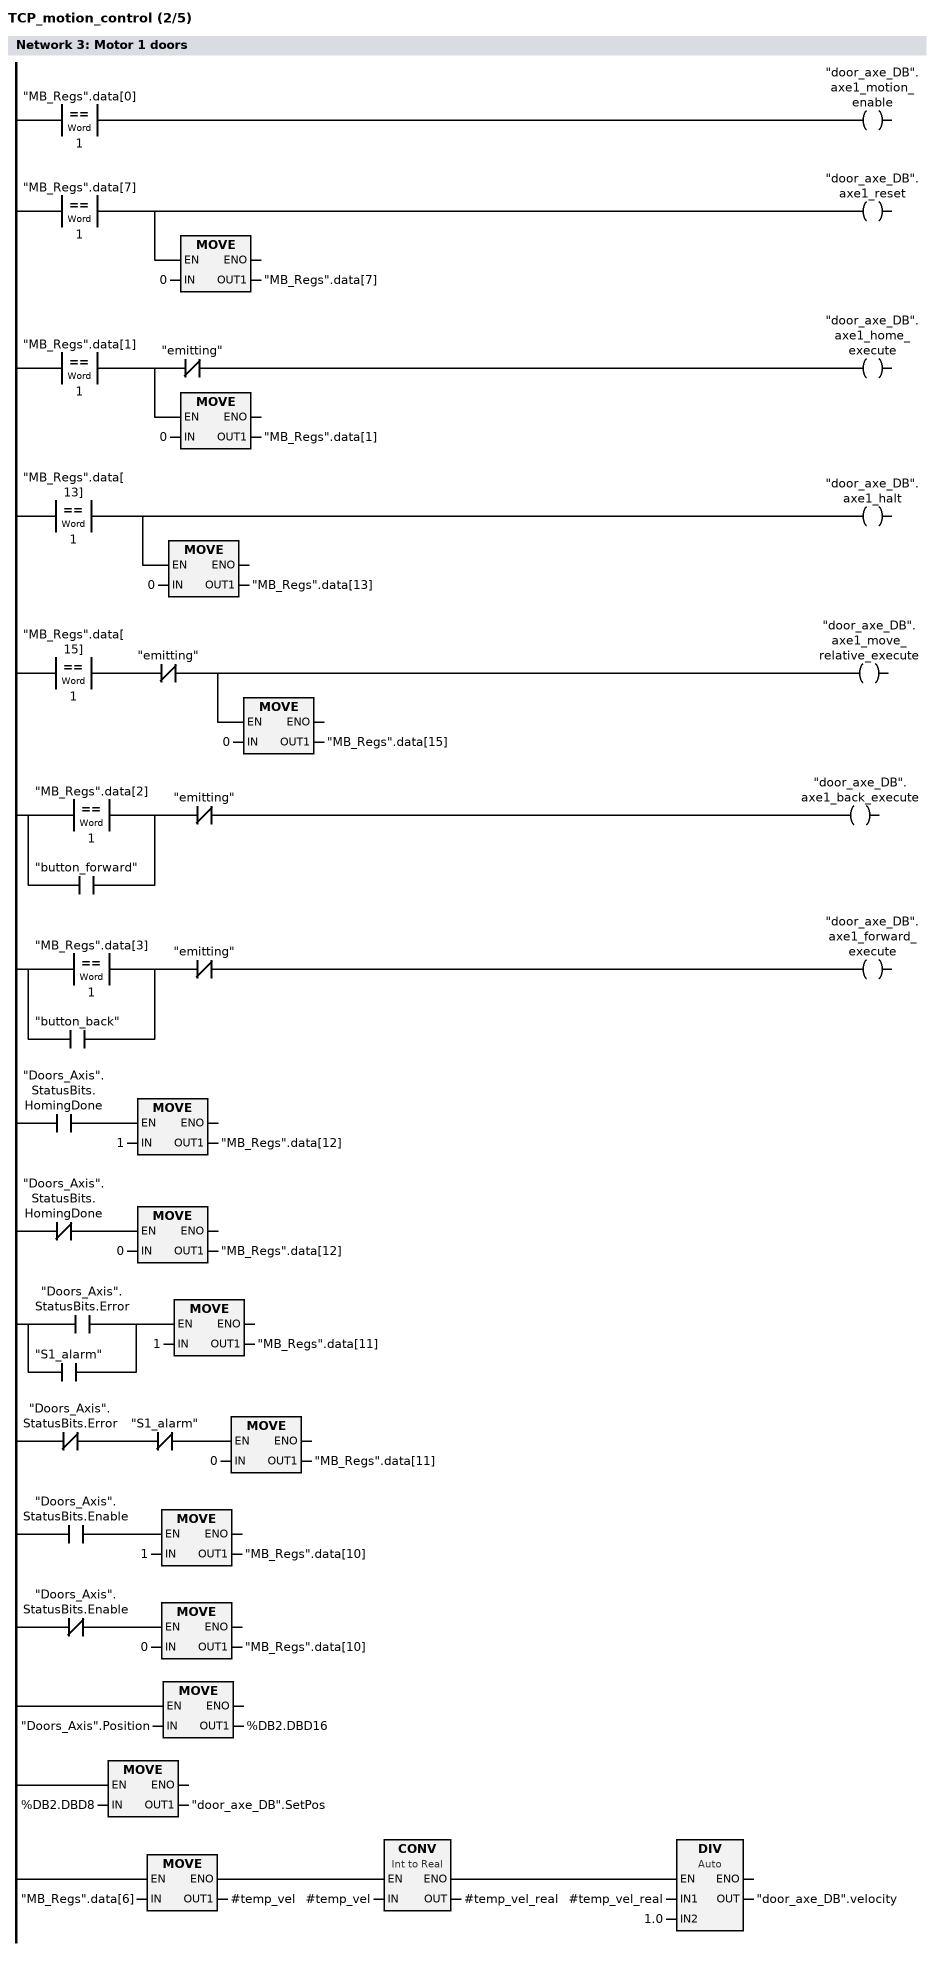
   RUNG wire#powerrail
      { S7_Templates := "SrcType := Word" } EQ_Contact(in1 := "MB_Regs".data[0], in2 := 1)
      Coil( "door_axe_DB".axe1_motion_enable )
   END_RUNG
   RUNG wire#powerrail
      { S7_Templates := "SrcType := Word" } EQ_Contact(in1 := "MB_Regs".data[7], in2 := 1)
      wire#w1
      Coil( "door_axe_DB".axe1_reset )
   END_RUNG
   RUNG wire#w1
      Move(in := 0, out1 => "MB_Regs".data[7])
   END_RUNG
   RUNG wire#powerrail
      { S7_Templates := "SrcType := Word" } EQ_Contact(in1 := "MB_Regs".data[1], in2 := 1)
      wire#w2
      I_Contact( "emitting" )
      Coil( "door_axe_DB".axe1_home_execute )
   END_RUNG
   RUNG wire#w2
      Move(in := 0, out1 => "MB_Regs".data[1])
   END_RUNG
   RUNG wire#powerrail
      { S7_Templates := "SrcType := Word" } EQ_Contact(in1 := "MB_Regs".data[13], in2 := 1)
      wire#w3
      Coil( "door_axe_DB".axe1_halt )
   END_RUNG
   RUNG wire#w3
      Move(in := 0, out1 => "MB_Regs".data[13])
   END_RUNG
   RUNG wire#powerrail
      { S7_Templates := "SrcType := Word" } EQ_Contact(in1 := "MB_Regs".data[15], in2 := 1)
      I_Contact( "emitting" )
      wire#w4
      Coil( "door_axe_DB".axe1_move_relative_execute )
   END_RUNG
   RUNG wire#w4
      Move(in := 0, out1 => "MB_Regs".data[15])
   END_RUNG
   RUNG wire#powerrail
      { S7_Templates := "SrcType := Word" } EQ_Contact(in1 := "MB_Regs".data[2], in2 := 1)
      wire#w5
      I_Contact( "emitting" )
      Coil( "door_axe_DB".axe1_back_execute )
   END_RUNG
   RUNG wire#powerrail
      Contact( "button_forward" )
   END_RUNG wire#w5
   RUNG wire#powerrail
      { S7_Templates := "SrcType := Word" } EQ_Contact(in1 := "MB_Regs".data[3], in2 := 1)
      wire#w6
      I_Contact( "emitting" )
      Coil( "door_axe_DB".axe1_forward_execute )
   END_RUNG
   RUNG wire#powerrail
      Contact( "button_back" )
   END_RUNG wire#w6
   RUNG wire#powerrail
      Contact( "Doors_Axis".StatusBits.HomingDone )
      Move(in := 1, out1 => "MB_Regs".data[12])
   END_RUNG
   RUNG wire#powerrail
      I_Contact( "Doors_Axis".StatusBits.HomingDone )
      Move(in := 0, out1 => "MB_Regs".data[12])
   END_RUNG
   RUNG wire#powerrail
      Contact( "Doors_Axis".StatusBits.Error )
      wire#w7
      Move(in := 1, out1 => "MB_Regs".data[11])
   END_RUNG
   RUNG wire#powerrail
      Contact( "S1_alarm" )
   END_RUNG wire#w7
   RUNG wire#powerrail
      I_Contact( "Doors_Axis".StatusBits.Error )
      I_Contact( "S1_alarm" )
      Move(in := 0, out1 => "MB_Regs".data[11])
   END_RUNG
   RUNG wire#powerrail
      Contact( "Doors_Axis".StatusBits.Enable )
      Move(in := 1, out1 => "MB_Regs".data[10])
   END_RUNG
   RUNG wire#powerrail
      I_Contact( "Doors_Axis".StatusBits.Enable )
      Move(in := 0, out1 => "MB_Regs".data[10])
   END_RUNG
   RUNG wire#powerrail
      Move(in := "Doors_Axis".Position, out1 => %DB2.DBD16)
   END_RUNG
   RUNG wire#powerrail
      Move(in := %DB2.DBD8, out1 => "door_axe_DB".SetPos)
   END_RUNG
   RUNG wire#powerrail
      Move(in := "MB_Regs".data[6], out1 => #temp_vel)
      { S7_Templates := "[SrcType := Int, DestType := Real]" } Convert(in := #temp_vel, out => #temp_vel_real)
      Div(in1 := #temp_vel_real, in2 := 1.0, out => "door_axe_DB".velocity)
   END_RUNG
   // the same network as SCL:
   "door_axe_DB".axe1_motion_enable := "MB_Regs".data[0] = 1;
   "door_axe_DB".axe1_reset := "MB_Regs".data[7] = 1;
   IF "door_axe_DB".axe1_reset THEN "MB_Regs".data[7] := 0; END_IF;
   #_w1 := "MB_Regs".data[1] = 1;
   "door_axe_DB".axe1_home_execute := #_w1 AND NOT "emitting";
   IF #_w1 THEN "MB_Regs".data[1] := 0; END_IF;
   "door_axe_DB".axe1_halt := "MB_Regs".data[13] = 1;
   IF "door_axe_DB".axe1_halt THEN "MB_Regs".data[13] := 0; END_IF;
   "door_axe_DB".axe1_move_relative_execute := ("MB_Regs".data[15] = 1) AND NOT "emitting";
   IF "door_axe_DB".axe1_move_relative_execute THEN "MB_Regs".data[15] := 0; END_IF;
   "door_axe_DB".axe1_back_execute := (("MB_Regs".data[2] = 1) OR "button_forward") AND NOT "emitting";
   "door_axe_DB".axe1_forward_execute := (("MB_Regs".data[3] = 1) OR "button_back") AND NOT "emitting";
   IF "Doors_Axis".StatusBits.HomingDone THEN "MB_Regs".data[12] := 1; END_IF;
   IF NOT "Doors_Axis".StatusBits.HomingDone THEN "MB_Regs".data[12] := 0; END_IF;
   IF "Doors_Axis".StatusBits.Error OR "S1_alarm" THEN "MB_Regs".data[11] := 1; END_IF;
   IF NOT "Doors_Axis".StatusBits.Error AND NOT "S1_alarm" THEN "MB_Regs".data[11] := 0; END_IF;
   IF "Doors_Axis".StatusBits.Enable THEN "MB_Regs".data[10] := 1; END_IF;
   IF NOT "Doors_Axis".StatusBits.Enable THEN "MB_Regs".data[10] := 0; END_IF;
   %DB2.DBD16 := "Doors_Axis".Position;
   "door_axe_DB".SetPos := %DB2.DBD8;
   #temp_vel := "MB_Regs".data[6];
   #temp_vel_real := INT_TO_REAL(#temp_vel);
   "door_axe_DB".velocity := #temp_vel_real / 1.0;
END_REGION

REGION Network 4: Motor 2 rotation
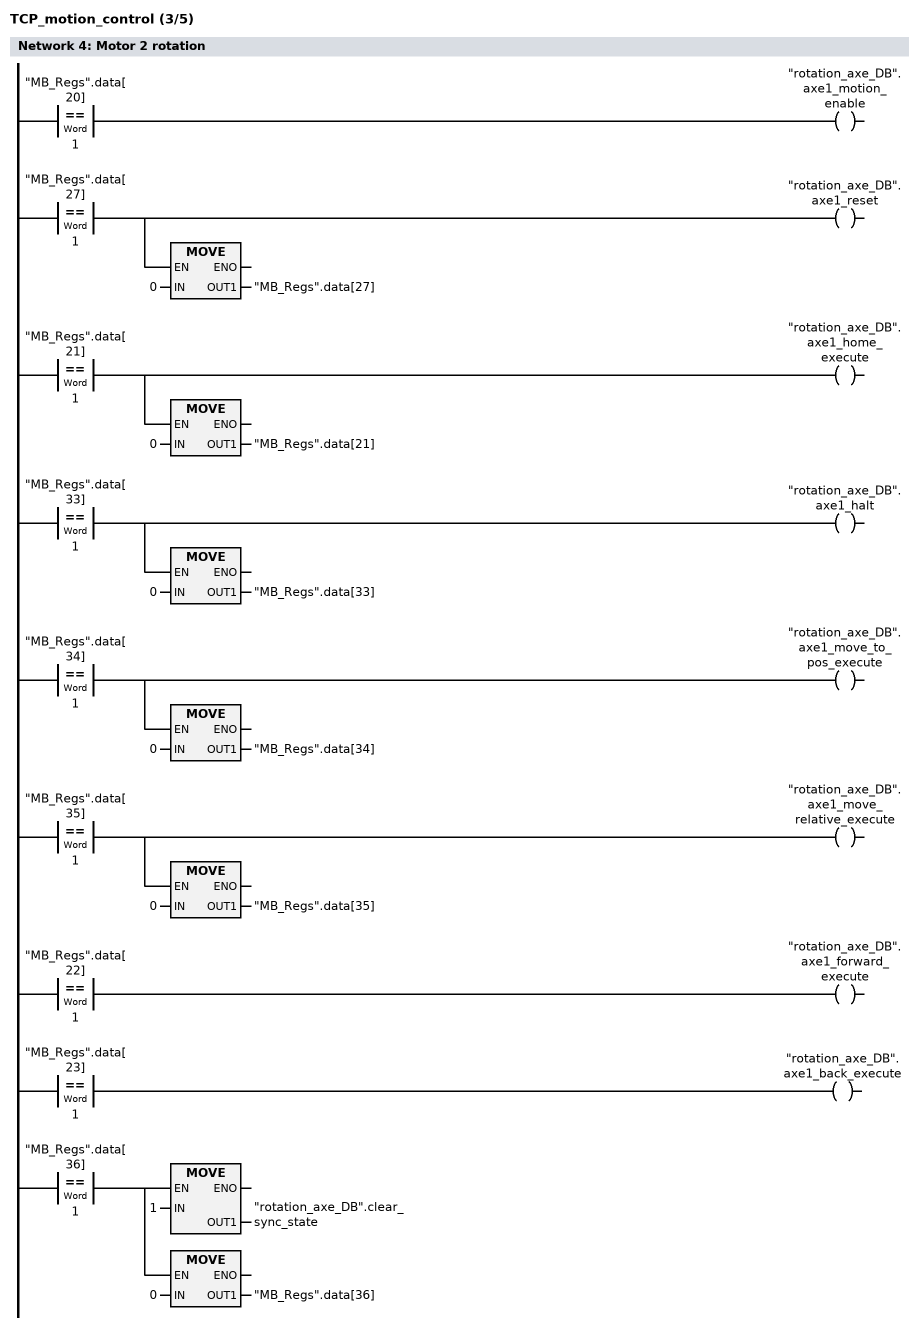
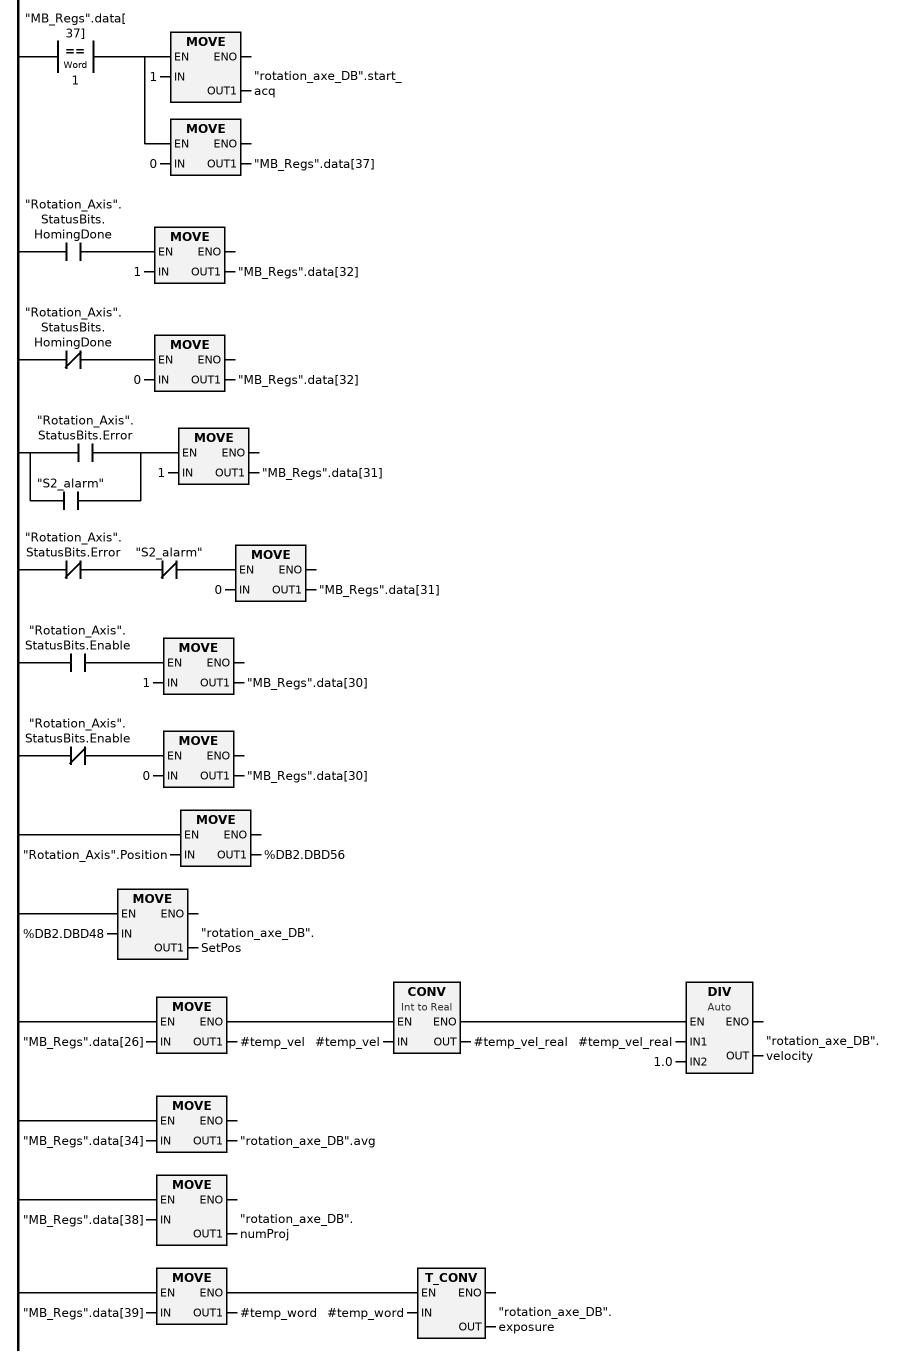
   "rotation_axe_DB".axe1_motion_enable := "MB_Regs".data[20] = 1;
   "rotation_axe_DB".axe1_reset := "MB_Regs".data[27] = 1;
   IF "rotation_axe_DB".axe1_reset THEN "MB_Regs".data[27] := 0; END_IF;
   "rotation_axe_DB".axe1_home_execute := "MB_Regs".data[21] = 1;
   IF "rotation_axe_DB".axe1_home_execute THEN "MB_Regs".data[21] := 0; END_IF;
   "rotation_axe_DB".axe1_halt := "MB_Regs".data[33] = 1;
   IF "rotation_axe_DB".axe1_halt THEN "MB_Regs".data[33] := 0; END_IF;
   "rotation_axe_DB".axe1_move_to_pos_execute := "MB_Regs".data[34] = 1;
   IF "rotation_axe_DB".axe1_move_to_pos_execute THEN "MB_Regs".data[34] := 0; END_IF;
   "rotation_axe_DB".axe1_move_relative_execute := "MB_Regs".data[35] = 1;
   IF "rotation_axe_DB".axe1_move_relative_execute THEN "MB_Regs".data[35] := 0; END_IF;
   "rotation_axe_DB".axe1_forward_execute := "MB_Regs".data[22] = 1;
   "rotation_axe_DB".axe1_back_execute := "MB_Regs".data[23] = 1;
   IF "MB_Regs".data[36] = 1 THEN
       "rotation_axe_DB".clear_sync_state := 1;
       "MB_Regs".data[36] := 0;
   END_IF;
   IF "MB_Regs".data[37] = 1 THEN
       "rotation_axe_DB".start_acq := 1;
       "MB_Regs".data[37] := 0;
   END_IF;
   IF "Rotation_Axis".StatusBits.HomingDone THEN "MB_Regs".data[32] := 1; END_IF;
   IF NOT "Rotation_Axis".StatusBits.HomingDone THEN "MB_Regs".data[32] := 0; END_IF;
   IF "Rotation_Axis".StatusBits.Error OR "S2_alarm" THEN "MB_Regs".data[31] := 1; END_IF;
   IF NOT "Rotation_Axis".StatusBits.Error AND NOT "S2_alarm" THEN "MB_Regs".data[31] := 0; END_IF;
   IF "Rotation_Axis".StatusBits.Enable THEN "MB_Regs".data[30] := 1; END_IF;
   IF NOT "Rotation_Axis".StatusBits.Enable THEN "MB_Regs".data[30] := 0; END_IF;
   %DB2.DBD56 := "Rotation_Axis".Position;
   "rotation_axe_DB".SetPos := %DB2.DBD48;
   #temp_vel := "MB_Regs".data[26];
   #temp_vel_real := INT_TO_REAL(#temp_vel);
   "rotation_axe_DB".velocity := #temp_vel_real / 1.0;
   "rotation_axe_DB".avg := "MB_Regs".data[34];
   "rotation_axe_DB".numProj := "MB_Regs".data[38];
   #temp_word := "MB_Regs".data[39];
   "rotation_axe_DB".exposure := T_CONV(IN := #temp_word);
END_REGION

REGION Network 5: Motor 3 (ISO)
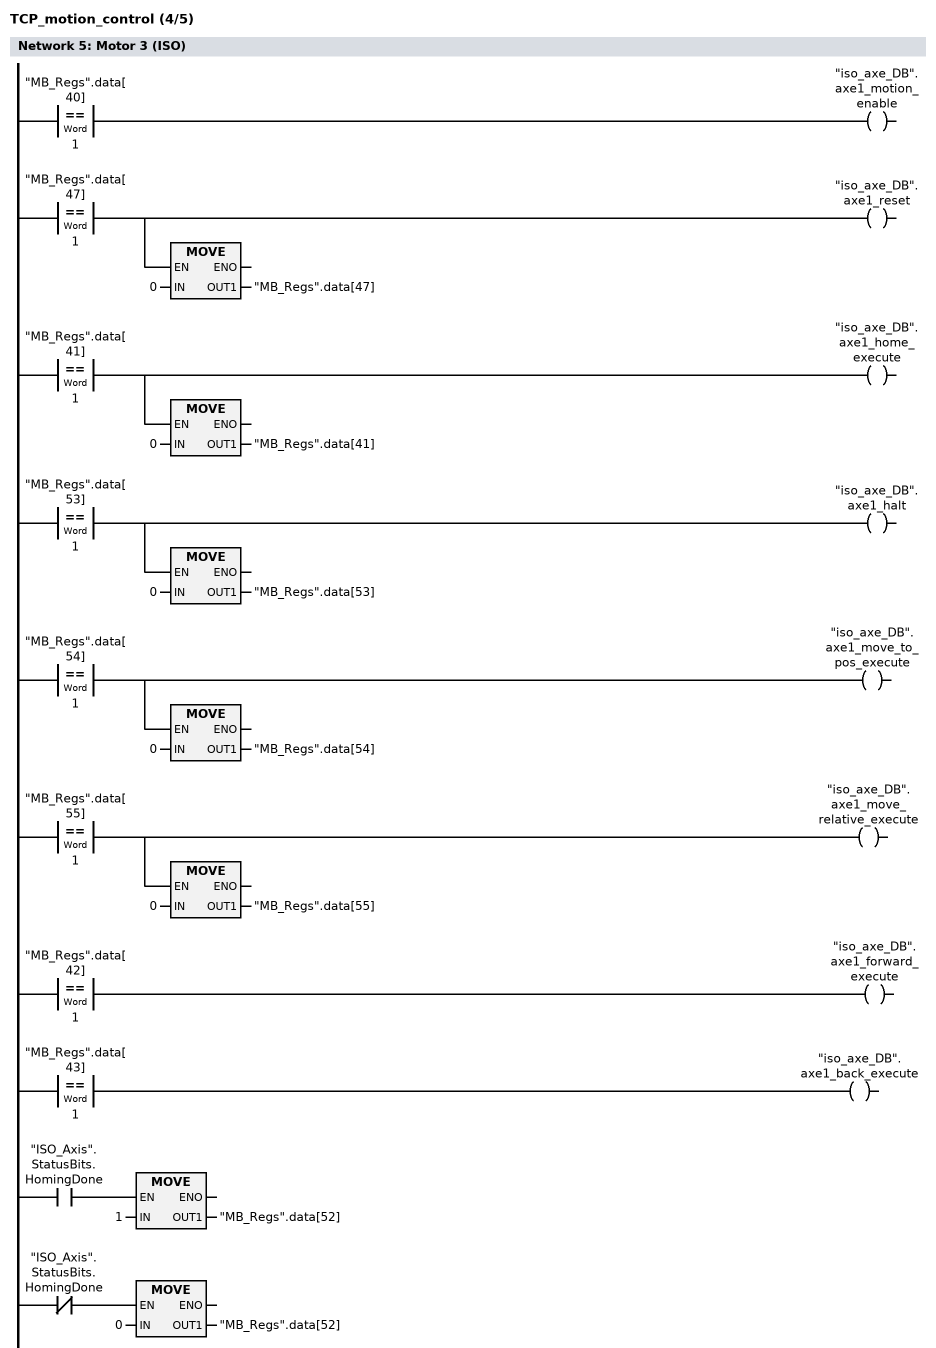
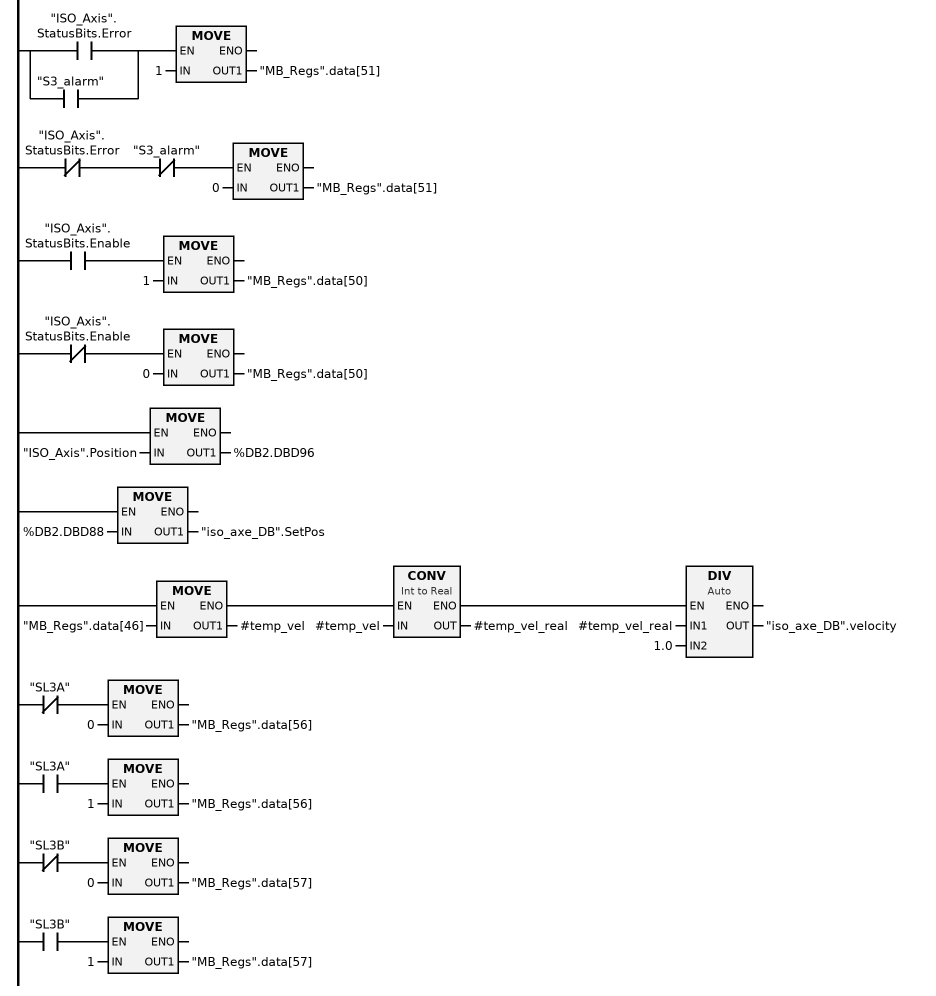
   RUNG wire#powerrail
      { S7_Templates := "SrcType := Word" } EQ_Contact(in1 := "MB_Regs".data[40], in2 := 1)
      Coil( "iso_axe_DB".axe1_motion_enable )
   END_RUNG
   RUNG wire#powerrail
      { S7_Templates := "SrcType := Word" } EQ_Contact(in1 := "MB_Regs".data[47], in2 := 1)
      wire#w1
      Coil( "iso_axe_DB".axe1_reset )
   END_RUNG
   RUNG wire#w1
      Move(in := 0, out1 => "MB_Regs".data[47])
   END_RUNG
   RUNG wire#powerrail
      { S7_Templates := "SrcType := Word" } EQ_Contact(in1 := "MB_Regs".data[41], in2 := 1)
      wire#w2
      Coil( "iso_axe_DB".axe1_home_execute )
   END_RUNG
   RUNG wire#w2
      Move(in := 0, out1 => "MB_Regs".data[41])
   END_RUNG
   RUNG wire#powerrail
      { S7_Templates := "SrcType := Word" } EQ_Contact(in1 := "MB_Regs".data[53], in2 := 1)
      wire#w3
      Coil( "iso_axe_DB".axe1_halt )
   END_RUNG
   RUNG wire#w3
      Move(in := 0, out1 => "MB_Regs".data[53])
   END_RUNG
   RUNG wire#powerrail
      { S7_Templates := "SrcType := Word" } EQ_Contact(in1 := "MB_Regs".data[54], in2 := 1)
      wire#w4
      Coil( "iso_axe_DB".axe1_move_to_pos_execute )
   END_RUNG
   RUNG wire#w4
      Move(in := 0, out1 => "MB_Regs".data[54])
   END_RUNG
   RUNG wire#powerrail
      { S7_Templates := "SrcType := Word" } EQ_Contact(in1 := "MB_Regs".data[55], in2 := 1)
      wire#w5
      Coil( "iso_axe_DB".axe1_move_relative_execute )
   END_RUNG
   RUNG wire#w5
      Move(in := 0, out1 => "MB_Regs".data[55])
   END_RUNG
   RUNG wire#powerrail
      { S7_Templates := "SrcType := Word" } EQ_Contact(in1 := "MB_Regs".data[42], in2 := 1)
      Coil( "iso_axe_DB".axe1_forward_execute )
   END_RUNG
   RUNG wire#powerrail
      { S7_Templates := "SrcType := Word" } EQ_Contact(in1 := "MB_Regs".data[43], in2 := 1)
      Coil( "iso_axe_DB".axe1_back_execute )
   END_RUNG
   RUNG wire#powerrail
      Contact( "ISO_Axis".StatusBits.HomingDone )
      Move(in := 1, out1 => "MB_Regs".data[52])
   END_RUNG
   RUNG wire#powerrail
      I_Contact( "ISO_Axis".StatusBits.HomingDone )
      Move(in := 0, out1 => "MB_Regs".data[52])
   END_RUNG
   RUNG wire#powerrail
      Contact( "ISO_Axis".StatusBits.Error )
      wire#w6
      Move(in := 1, out1 => "MB_Regs".data[51])
   END_RUNG
   RUNG wire#powerrail
      Contact( "S3_alarm" )
   END_RUNG wire#w6
   RUNG wire#powerrail
      I_Contact( "ISO_Axis".StatusBits.Error )
      I_Contact( "S3_alarm" )
      Move(in := 0, out1 => "MB_Regs".data[51])
   END_RUNG
   RUNG wire#powerrail
      Contact( "ISO_Axis".StatusBits.Enable )
      Move(in := 1, out1 => "MB_Regs".data[50])
   END_RUNG
   RUNG wire#powerrail
      I_Contact( "ISO_Axis".StatusBits.Enable )
      Move(in := 0, out1 => "MB_Regs".data[50])
   END_RUNG
   RUNG wire#powerrail
      Move(in := "ISO_Axis".Position, out1 => %DB2.DBD96)
   END_RUNG
   RUNG wire#powerrail
      Move(in := %DB2.DBD88, out1 => "iso_axe_DB".SetPos)
   END_RUNG
   RUNG wire#powerrail
      Move(in := "MB_Regs".data[46], out1 => #temp_vel)
      { S7_Templates := "[SrcType := Int, DestType := Real]" } Convert(in := #temp_vel, out => #temp_vel_real)
      Div(in1 := #temp_vel_real, in2 := 1.0, out => "iso_axe_DB".velocity)
   END_RUNG
   RUNG wire#powerrail
      I_Contact( "SL3A" )
      Move(in := 0, out1 => "MB_Regs".data[56])
   END_RUNG
   RUNG wire#powerrail
      Contact( "SL3A" )
      Move(in := 1, out1 => "MB_Regs".data[56])
   END_RUNG
   RUNG wire#powerrail
      I_Contact( "SL3B" )
      Move(in := 0, out1 => "MB_Regs".data[57])
   END_RUNG
   RUNG wire#powerrail
      Contact( "SL3B" )
      Move(in := 1, out1 => "MB_Regs".data[57])
   END_RUNG
   // the same network as SCL:
   "iso_axe_DB".axe1_motion_enable := "MB_Regs".data[40] = 1;
   "iso_axe_DB".axe1_reset := "MB_Regs".data[47] = 1;
   IF "iso_axe_DB".axe1_reset THEN "MB_Regs".data[47] := 0; END_IF;
   "iso_axe_DB".axe1_home_execute := "MB_Regs".data[41] = 1;
   IF "iso_axe_DB".axe1_home_execute THEN "MB_Regs".data[41] := 0; END_IF;
   "iso_axe_DB".axe1_halt := "MB_Regs".data[53] = 1;
   IF "iso_axe_DB".axe1_halt THEN "MB_Regs".data[53] := 0; END_IF;
   "iso_axe_DB".axe1_move_to_pos_execute := "MB_Regs".data[54] = 1;
   IF "iso_axe_DB".axe1_move_to_pos_execute THEN "MB_Regs".data[54] := 0; END_IF;
   "iso_axe_DB".axe1_move_relative_execute := "MB_Regs".data[55] = 1;
   IF "iso_axe_DB".axe1_move_relative_execute THEN "MB_Regs".data[55] := 0; END_IF;
   "iso_axe_DB".axe1_forward_execute := "MB_Regs".data[42] = 1;
   "iso_axe_DB".axe1_back_execute := "MB_Regs".data[43] = 1;
   IF "ISO_Axis".StatusBits.HomingDone THEN "MB_Regs".data[52] := 1; END_IF;
   IF NOT "ISO_Axis".StatusBits.HomingDone THEN "MB_Regs".data[52] := 0; END_IF;
   IF "ISO_Axis".StatusBits.Error OR "S3_alarm" THEN "MB_Regs".data[51] := 1; END_IF;
   IF NOT "ISO_Axis".StatusBits.Error AND NOT "S3_alarm" THEN "MB_Regs".data[51] := 0; END_IF;
   IF "ISO_Axis".StatusBits.Enable THEN "MB_Regs".data[50] := 1; END_IF;
   IF NOT "ISO_Axis".StatusBits.Enable THEN "MB_Regs".data[50] := 0; END_IF;
   %DB2.DBD96 := "ISO_Axis".Position;
   "iso_axe_DB".SetPos := %DB2.DBD88;
   #temp_vel := "MB_Regs".data[46];
   #temp_vel_real := INT_TO_REAL(#temp_vel);
   "iso_axe_DB".velocity := #temp_vel_real / 1.0;
   IF NOT "SL3A" THEN "MB_Regs".data[56] := 0; END_IF;
   IF "SL3A" THEN "MB_Regs".data[56] := 1; END_IF;
   IF NOT "SL3B" THEN "MB_Regs".data[57] := 0; END_IF;
   IF "SL3B" THEN "MB_Regs".data[57] := 1; END_IF;
END_REGION

REGION Network 6: Motor 4 (Detector)
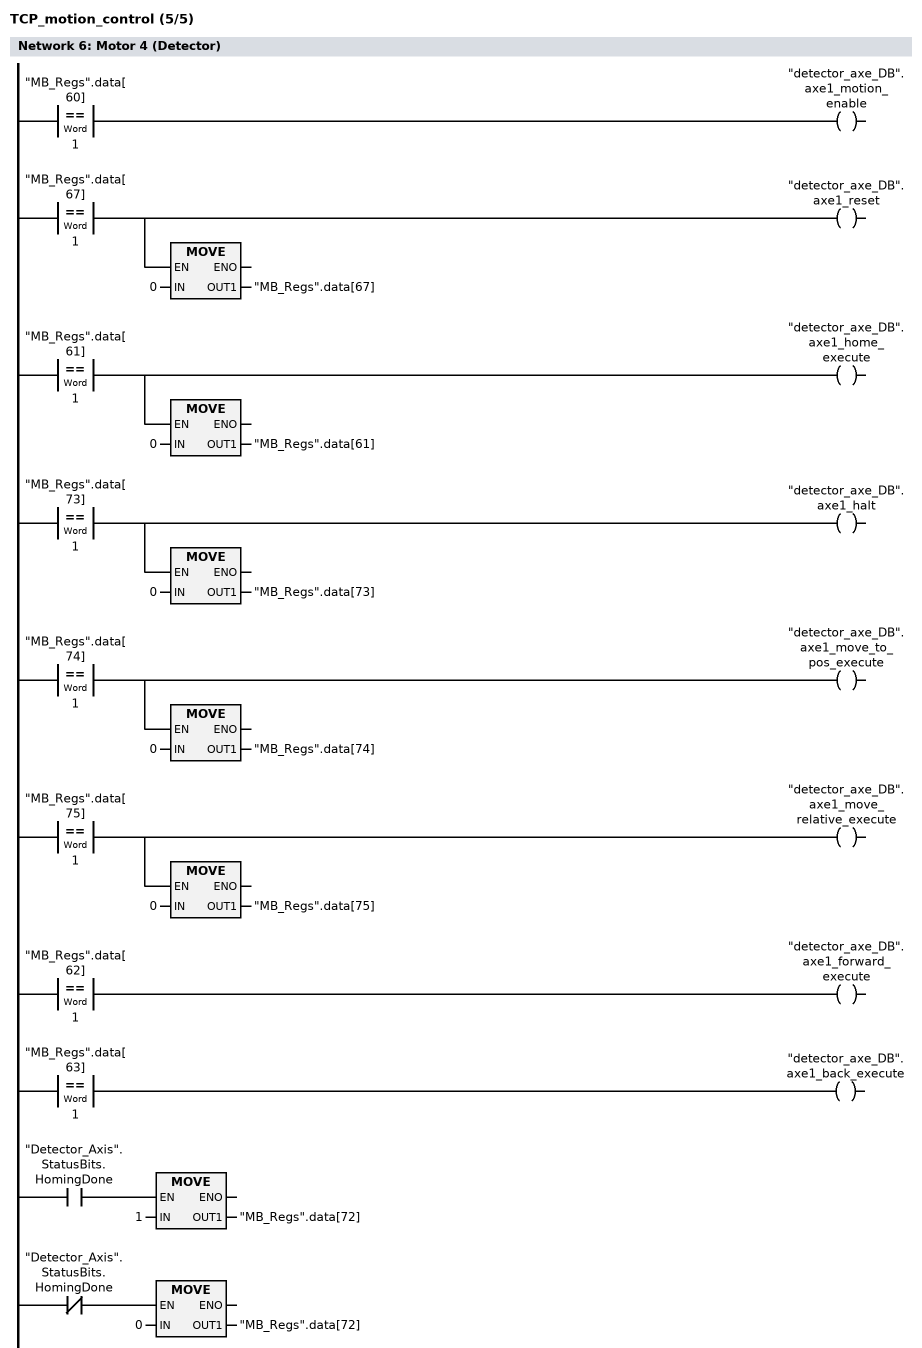
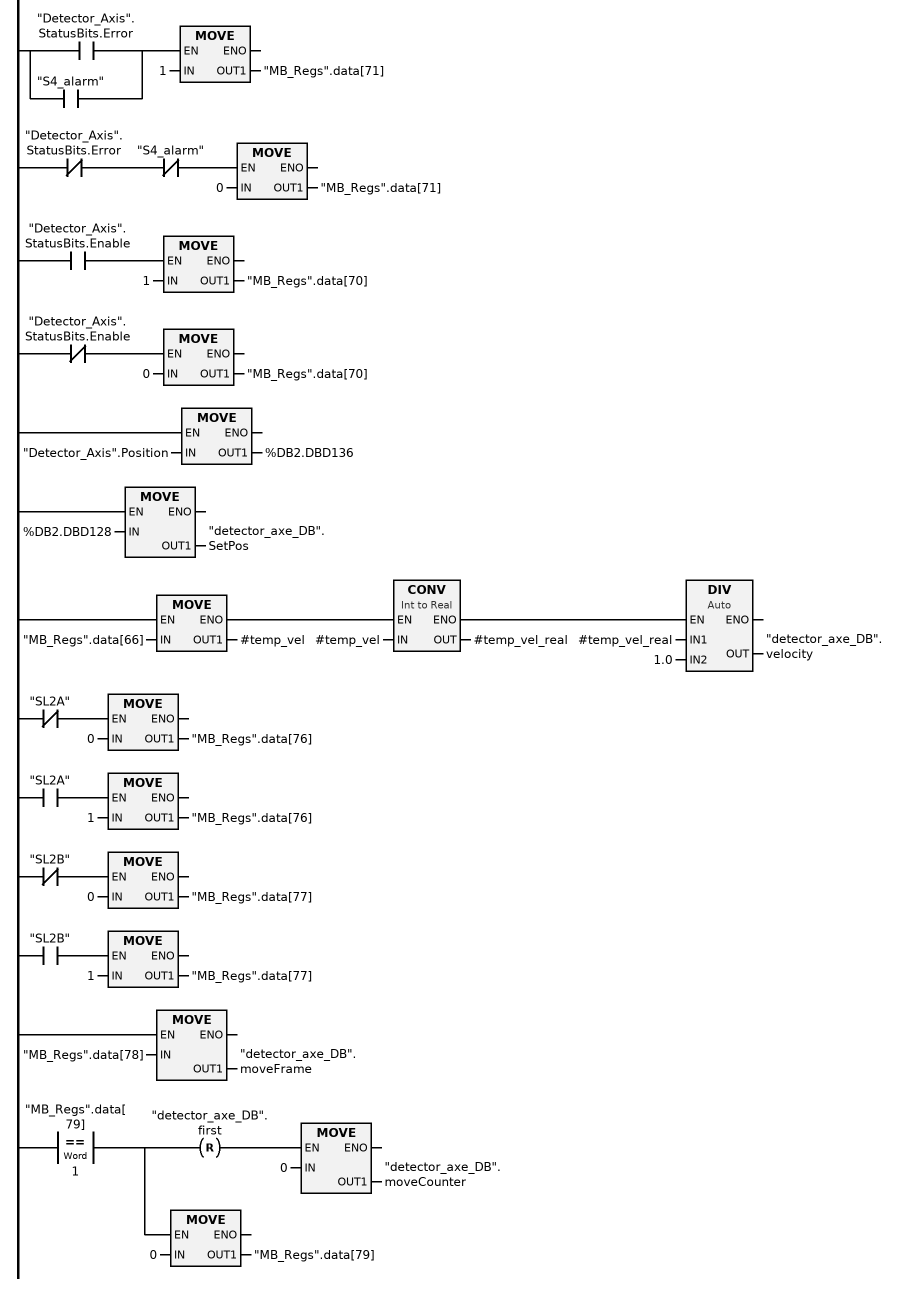
   RUNG wire#powerrail
      { S7_Templates := "SrcType := Word" } EQ_Contact(in1 := "MB_Regs".data[60], in2 := 1)
      Coil( "detector_axe_DB".axe1_motion_enable )
   END_RUNG
   RUNG wire#powerrail
      { S7_Templates := "SrcType := Word" } EQ_Contact(in1 := "MB_Regs".data[67], in2 := 1)
      wire#w1
      Coil( "detector_axe_DB".axe1_reset )
   END_RUNG
   RUNG wire#w1
      Move(in := 0, out1 => "MB_Regs".data[67])
   END_RUNG
   RUNG wire#powerrail
      { S7_Templates := "SrcType := Word" } EQ_Contact(in1 := "MB_Regs".data[61], in2 := 1)
      wire#w2
      Coil( "detector_axe_DB".axe1_home_execute )
   END_RUNG
   RUNG wire#w2
      Move(in := 0, out1 => "MB_Regs".data[61])
   END_RUNG
   RUNG wire#powerrail
      { S7_Templates := "SrcType := Word" } EQ_Contact(in1 := "MB_Regs".data[73], in2 := 1)
      wire#w3
      Coil( "detector_axe_DB".axe1_halt )
   END_RUNG
   RUNG wire#w3
      Move(in := 0, out1 => "MB_Regs".data[73])
   END_RUNG
   RUNG wire#powerrail
      { S7_Templates := "SrcType := Word" } EQ_Contact(in1 := "MB_Regs".data[74], in2 := 1)
      wire#w4
      Coil( "detector_axe_DB".axe1_move_to_pos_execute )
   END_RUNG
   RUNG wire#w4
      Move(in := 0, out1 => "MB_Regs".data[74])
   END_RUNG
   RUNG wire#powerrail
      { S7_Templates := "SrcType := Word" } EQ_Contact(in1 := "MB_Regs".data[75], in2 := 1)
      wire#w5
      Coil( "detector_axe_DB".axe1_move_relative_execute )
   END_RUNG
   RUNG wire#w5
      Move(in := 0, out1 => "MB_Regs".data[75])
   END_RUNG
   RUNG wire#powerrail
      { S7_Templates := "SrcType := Word" } EQ_Contact(in1 := "MB_Regs".data[62], in2 := 1)
      Coil( "detector_axe_DB".axe1_forward_execute )
   END_RUNG
   RUNG wire#powerrail
      { S7_Templates := "SrcType := Word" } EQ_Contact(in1 := "MB_Regs".data[63], in2 := 1)
      Coil( "detector_axe_DB".axe1_back_execute )
   END_RUNG
   RUNG wire#powerrail
      Contact( "Detector_Axis".StatusBits.HomingDone )
      Move(in := 1, out1 => "MB_Regs".data[72])
   END_RUNG
   RUNG wire#powerrail
      I_Contact( "Detector_Axis".StatusBits.HomingDone )
      Move(in := 0, out1 => "MB_Regs".data[72])
   END_RUNG
   RUNG wire#powerrail
      Contact( "Detector_Axis".StatusBits.Error )
      wire#w6
      Move(in := 1, out1 => "MB_Regs".data[71])
   END_RUNG
   RUNG wire#powerrail
      Contact( "S4_alarm" )
   END_RUNG wire#w6
   RUNG wire#powerrail
      I_Contact( "Detector_Axis".StatusBits.Error )
      I_Contact( "S4_alarm" )
      Move(in := 0, out1 => "MB_Regs".data[71])
   END_RUNG
   RUNG wire#powerrail
      Contact( "Detector_Axis".StatusBits.Enable )
      Move(in := 1, out1 => "MB_Regs".data[70])
   END_RUNG
   RUNG wire#powerrail
      I_Contact( "Detector_Axis".StatusBits.Enable )
      Move(in := 0, out1 => "MB_Regs".data[70])
   END_RUNG
   RUNG wire#powerrail
      Move(in := "Detector_Axis".Position, out1 => %DB2.DBD136)
   END_RUNG
   RUNG wire#powerrail
      Move(in := %DB2.DBD128, out1 => "detector_axe_DB".SetPos)
   END_RUNG
   RUNG wire#powerrail
      Move(in := "MB_Regs".data[66], out1 => #temp_vel)
      { S7_Templates := "[SrcType := Int, DestType := Real]" } Convert(in := #temp_vel, out => #temp_vel_real)
      Div(in1 := #temp_vel_real, in2 := 1.0, out => "detector_axe_DB".velocity)
   END_RUNG
   RUNG wire#powerrail
      I_Contact( "SL2A" )
      Move(in := 0, out1 => "MB_Regs".data[76])
   END_RUNG
   RUNG wire#powerrail
      Contact( "SL2A" )
      Move(in := 1, out1 => "MB_Regs".data[76])
   END_RUNG
   RUNG wire#powerrail
      I_Contact( "SL2B" )
      Move(in := 0, out1 => "MB_Regs".data[77])
   END_RUNG
   RUNG wire#powerrail
      Contact( "SL2B" )
      Move(in := 1, out1 => "MB_Regs".data[77])
   END_RUNG
   RUNG wire#powerrail
      Move(in := "MB_Regs".data[78], out1 => "detector_axe_DB".moveFrame)
   END_RUNG
   RUNG wire#powerrail
      { S7_Templates := "SrcType := Word" } EQ_Contact(in1 := "MB_Regs".data[79], in2 := 1)
      wire#w7
      R_Coil( "detector_axe_DB".first )
      Move(in := 0, out1 => "detector_axe_DB".moveCounter)
   END_RUNG
   RUNG wire#w7
      Move(in := 0, out1 => "MB_Regs".data[79])
   END_RUNG
   // the same network as SCL:
   "detector_axe_DB".axe1_motion_enable := "MB_Regs".data[60] = 1;
   "detector_axe_DB".axe1_reset := "MB_Regs".data[67] = 1;
   IF "detector_axe_DB".axe1_reset THEN "MB_Regs".data[67] := 0; END_IF;
   "detector_axe_DB".axe1_home_execute := "MB_Regs".data[61] = 1;
   IF "detector_axe_DB".axe1_home_execute THEN "MB_Regs".data[61] := 0; END_IF;
   "detector_axe_DB".axe1_halt := "MB_Regs".data[73] = 1;
   IF "detector_axe_DB".axe1_halt THEN "MB_Regs".data[73] := 0; END_IF;
   "detector_axe_DB".axe1_move_to_pos_execute := "MB_Regs".data[74] = 1;
   IF "detector_axe_DB".axe1_move_to_pos_execute THEN "MB_Regs".data[74] := 0; END_IF;
   "detector_axe_DB".axe1_move_relative_execute := "MB_Regs".data[75] = 1;
   IF "detector_axe_DB".axe1_move_relative_execute THEN "MB_Regs".data[75] := 0; END_IF;
   "detector_axe_DB".axe1_forward_execute := "MB_Regs".data[62] = 1;
   "detector_axe_DB".axe1_back_execute := "MB_Regs".data[63] = 1;
   IF "Detector_Axis".StatusBits.HomingDone THEN "MB_Regs".data[72] := 1; END_IF;
   IF NOT "Detector_Axis".StatusBits.HomingDone THEN "MB_Regs".data[72] := 0; END_IF;
   IF "Detector_Axis".StatusBits.Error OR "S4_alarm" THEN "MB_Regs".data[71] := 1; END_IF;
   IF NOT "Detector_Axis".StatusBits.Error AND NOT "S4_alarm" THEN "MB_Regs".data[71] := 0; END_IF;
   IF "Detector_Axis".StatusBits.Enable THEN "MB_Regs".data[70] := 1; END_IF;
   IF NOT "Detector_Axis".StatusBits.Enable THEN "MB_Regs".data[70] := 0; END_IF;
   %DB2.DBD136 := "Detector_Axis".Position;
   "detector_axe_DB".SetPos := %DB2.DBD128;
   #temp_vel := "MB_Regs".data[66];
   #temp_vel_real := INT_TO_REAL(#temp_vel);
   "detector_axe_DB".velocity := #temp_vel_real / 1.0;
   IF NOT "SL2A" THEN "MB_Regs".data[76] := 0; END_IF;
   IF "SL2A" THEN "MB_Regs".data[76] := 1; END_IF;
   IF NOT "SL2B" THEN "MB_Regs".data[77] := 0; END_IF;
   IF "SL2B" THEN "MB_Regs".data[77] := 1; END_IF;
   "detector_axe_DB".moveFrame := "MB_Regs".data[78];
   IF "MB_Regs".data[79] = 1 THEN
       "detector_axe_DB".first := FALSE;
       "detector_axe_DB".moveCounter := 0;
       "MB_Regs".data[79] := 0;
   END_IF;
END_REGION
END_FUNCTION_BLOCK

FUNCTION_BLOCK "door_axe"   // FB2, LAD
{ S7_Optimized_Access := 'TRUE' }
VERSION : 0.1
   VAR
      SetPos : Real;
      velocity : Real;
      axe1_motion_enable : Bool;
      axe1_reset : Bool;
      axe1_halt : Bool;
      axe1_forward_execute : Bool;
      axe1_back_execute : Bool;
      axe1_home_execute : Bool;
      axe1_move_to_pos_execute : Bool;
      axe1_move_relative_execute : Bool;
      home_3_busy : Bool;
      home_0_busy : Bool;
      home_3_mode : Bool;
      home_0_mode : Bool;
      axe1_move_done : Bool;
      status : Bool;
   END_VAR
   VAR_TEMP
      temp_val2 : Real;
   END_VAR
   VAR CONSTANT
      vel_const : Real := 2.5;
   END_VAR
   VAR_TEMP   // added for the SCL form of the ladder/FBD networks
      _w1 : Bool;
   END_VAR
BEGIN

REGION Network 1
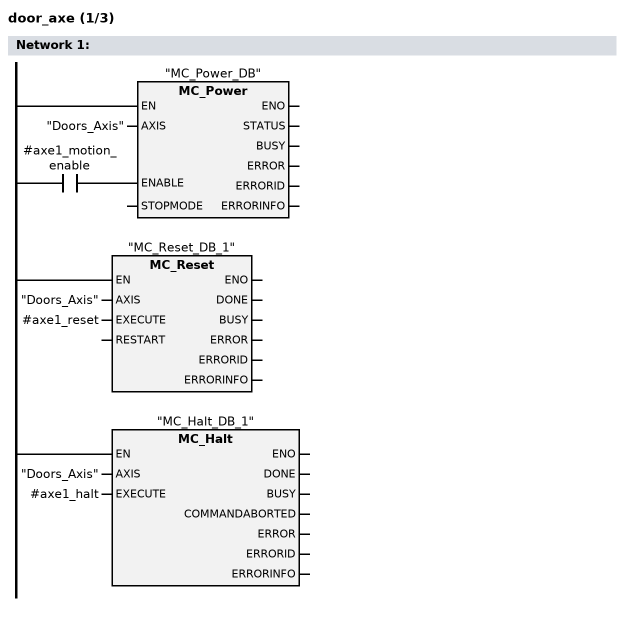
   "MC_Power_DB"(Axis := "Doors_Axis", Enable := #axe1_motion_enable);   // MC_Power
   "MC_Reset_DB_1"(Axis := "Doors_Axis", Execute := #axe1_reset);   // MC_Reset
   "MC_Halt_DB_1"(Axis := "Doors_Axis", Execute := #axe1_halt);   // MC_Halt
END_REGION

REGION Network 2
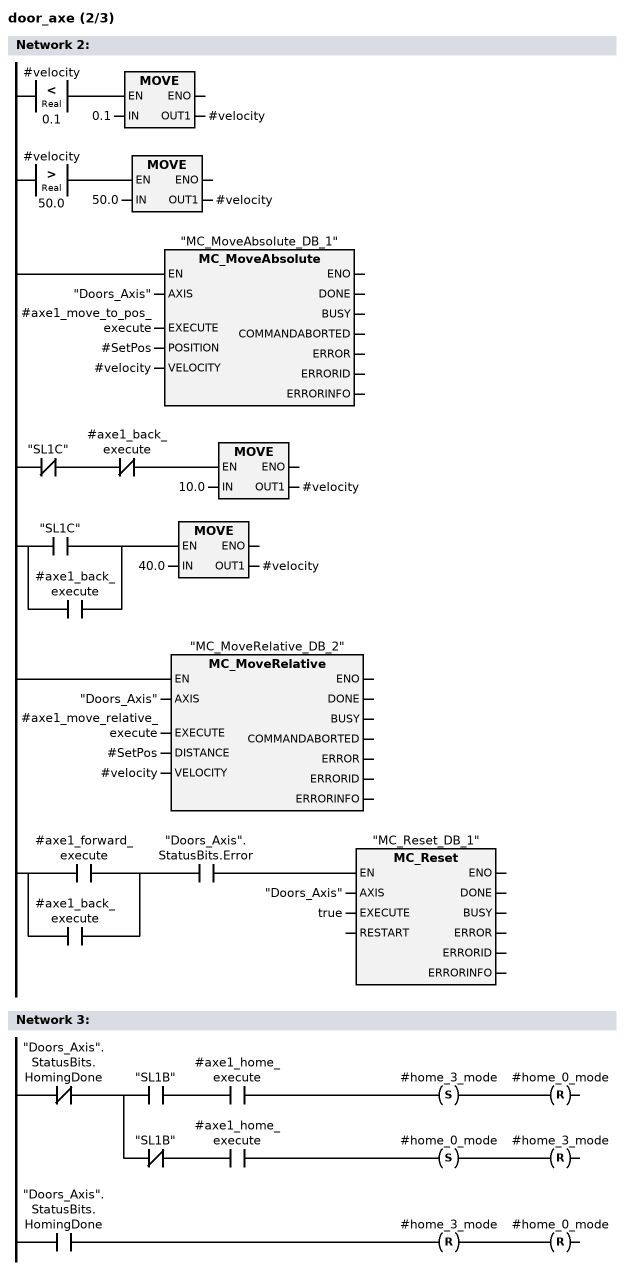
   IF #velocity < 0.1 THEN #velocity := 0.1; END_IF;
   IF #velocity > 50.0 THEN #velocity := 50.0; END_IF;
   "MC_MoveAbsolute_DB_1"(Axis := "Doors_Axis",   // MC_MoveAbsolute
                          Execute := #axe1_move_to_pos_execute,
                          Position := #SetPos,
                          Velocity := #velocity);
   IF NOT "SL1C" AND NOT #axe1_back_execute THEN #velocity := 10.0; END_IF;
   IF "SL1C" OR #axe1_back_execute THEN #velocity := 40.0; END_IF;
   "MC_MoveRelative_DB_2"(Axis := "Doors_Axis",   // MC_MoveRelative
                          Execute := #axe1_move_relative_execute,
                          Distance := #SetPos,
                          Velocity := #velocity);
   IF (#axe1_forward_execute OR #axe1_back_execute) AND "Doors_Axis".StatusBits.Error THEN
       "MC_Reset_DB_1"(Axis := "Doors_Axis", Execute := true);   // MC_Reset
   END_IF;
END_REGION

REGION Network 3
   RUNG wire#powerrail
      I_Contact( "Doors_Axis".StatusBits.HomingDone )
      wire#w1
      Contact( "SL1B" )
      Contact( #axe1_home_execute )
      S_Coil( #home_3_mode )
      R_Coil( #home_0_mode )
   END_RUNG
   RUNG wire#w1
      I_Contact( "SL1B" )
      Contact( #axe1_home_execute )
      S_Coil( #home_0_mode )
      R_Coil( #home_3_mode )
   END_RUNG
   RUNG wire#powerrail
      Contact( "Doors_Axis".StatusBits.HomingDone )
      R_Coil( #home_3_mode )
      R_Coil( #home_0_mode )
   END_RUNG
   // the same network as SCL:
   #_w1 := NOT "Doors_Axis".StatusBits.HomingDone;
   IF #_w1 AND "SL1B" AND #axe1_home_execute THEN
       #home_3_mode := TRUE;
       #home_0_mode := FALSE;
   END_IF;
   IF #_w1 AND NOT "SL1B" AND #axe1_home_execute THEN
       #home_0_mode := TRUE;
       #home_3_mode := FALSE;
   END_IF;
   IF "Doors_Axis".StatusBits.HomingDone THEN
       #home_3_mode := FALSE;
       #home_0_mode := FALSE;
   END_IF;
END_REGION

REGION Network 4: Ручная калибровка
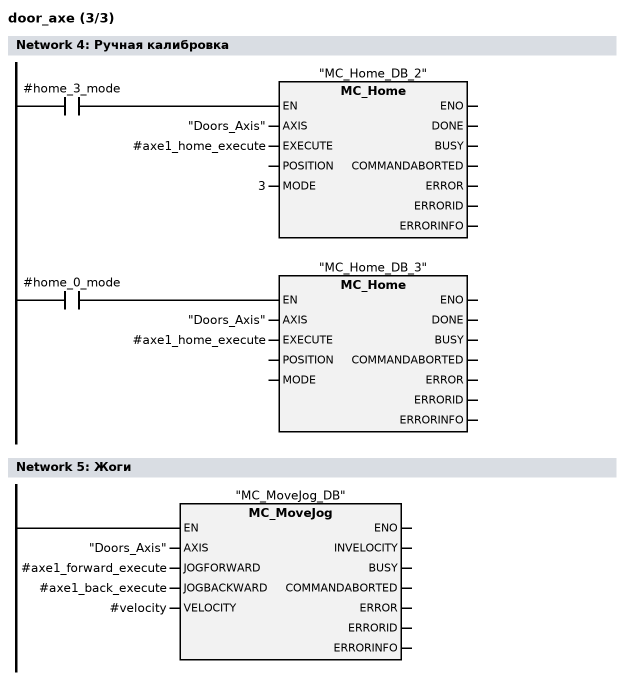
   IF #home_3_mode THEN
       "MC_Home_DB_2"(Axis := "Doors_Axis", Execute := #axe1_home_execute, Mode := 3);   // MC_Home
   END_IF;
   IF #home_0_mode THEN
       "MC_Home_DB_3"(Axis := "Doors_Axis", Execute := #axe1_home_execute);   // MC_Home
   END_IF;
END_REGION

REGION Network 5: Жоги
   "MC_MoveJog_DB"(Axis := "Doors_Axis",   // MC_MoveJog
                   JogForward := #axe1_forward_execute,
                   JogBackward := #axe1_back_execute,
                   Velocity := #velocity);
END_REGION
END_FUNCTION_BLOCK

FUNCTION_BLOCK "rotation_axe"   // FB3, LAD
{ S7_Optimized_Access := 'TRUE' }
VERSION : 0.1
   VAR
      SetPos : Real;
      velocity : Real;
      axe1_motion_enable : Bool;
      axe1_reset : Bool;
      axe1_halt : Bool;
      axe1_forward_execute : Bool;
      axe1_back_execute : Bool;
      axe1_home_execute : Bool;
      axe1_move_to_pos_execute : Bool;
      axe1_move_relative_execute : Bool;
      home_3_busy : Bool;
      home_0_busy : Bool;
      home_3_mode : Bool;
      home_0_mode : Bool;
      axe1_move_done : Bool;
      status : Bool;
      clear_sync_state : Word;
      start_acq : Word;
      projInd : Int;
      numProj : Word;
      exposure : Time;
      avg : Word;
      step1 : Word;
      step2 : Word;
      exposure_phase : Word;
      frd : Word;
      rot : Bool;
      busy : Bool;
      outTime_1 : DTL;
      outTime_12 : DTL;
      retTime_1 : Time;
      outTime_2 : DTL;
      outTime_22 : DTL;
      retTime_2 : Time;
      avgCounter : Word;
      ret : Int;
   END_VAR
   VAR CONSTANT
      vel_const : Real := 2.5;
   END_VAR
   VAR_TEMP   // added for the SCL form of the ladder/FBD networks
      _w1 : Bool;
      _w2 : Bool;
      _w3 : Bool;
      _w4 : Bool;
   END_VAR
BEGIN

REGION Network 1
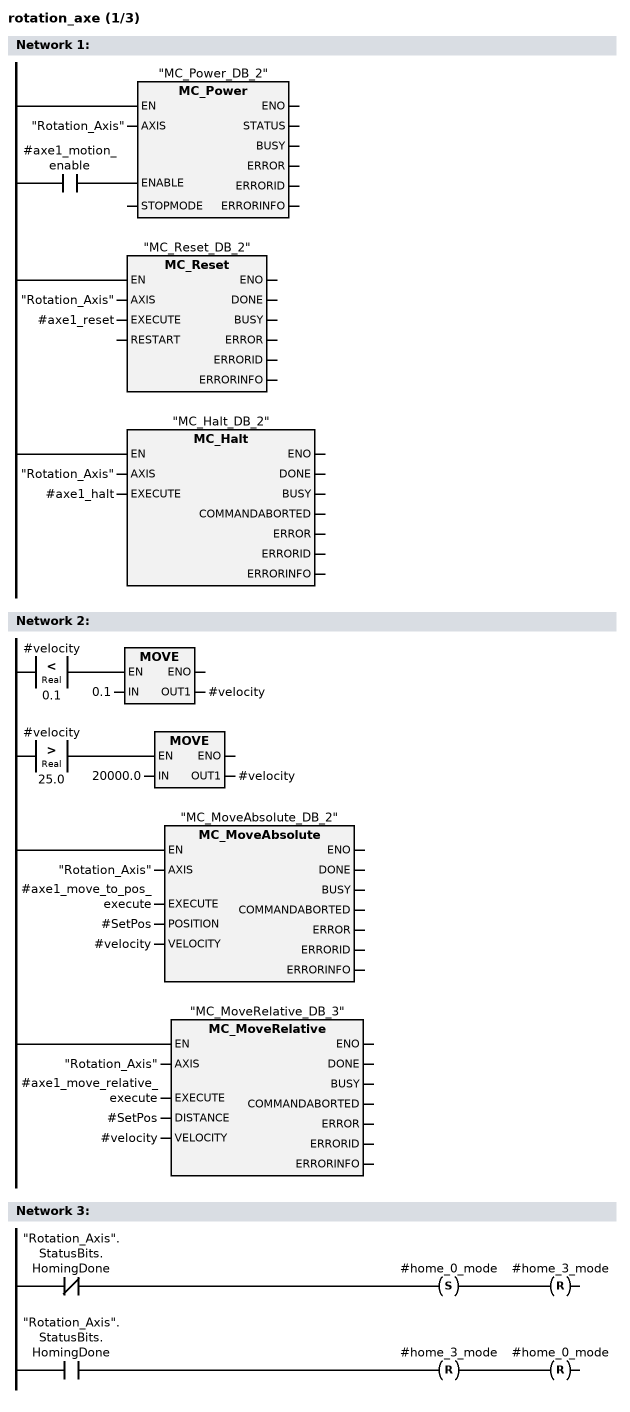
   "MC_Power_DB_2"(Axis := "Rotation_Axis", Enable := #axe1_motion_enable);   // MC_Power
   "MC_Reset_DB_2"(Axis := "Rotation_Axis", Execute := #axe1_reset);   // MC_Reset
   "MC_Halt_DB_2"(Axis := "Rotation_Axis", Execute := #axe1_halt);   // MC_Halt
END_REGION

REGION Network 2
   IF #velocity < 0.1 THEN #velocity := 0.1; END_IF;
   IF #velocity > 25.0 THEN #velocity := 20000.0; END_IF;
   "MC_MoveAbsolute_DB_2"(Axis := "Rotation_Axis",   // MC_MoveAbsolute
                          Execute := #axe1_move_to_pos_execute,
                          Position := #SetPos,
                          Velocity := #velocity);
   "MC_MoveRelative_DB_3"(Axis := "Rotation_Axis",   // MC_MoveRelative
                          Execute := #axe1_move_relative_execute,
                          Distance := #SetPos,
                          Velocity := #velocity);
END_REGION

REGION Network 3
   RUNG wire#powerrail
      I_Contact( "Rotation_Axis".StatusBits.HomingDone )
      S_Coil( #home_0_mode )
      R_Coil( #home_3_mode )
   END_RUNG
   RUNG wire#powerrail
      Contact( "Rotation_Axis".StatusBits.HomingDone )
      R_Coil( #home_3_mode )
      R_Coil( #home_0_mode )
   END_RUNG
   // the same network as SCL:
   IF NOT "Rotation_Axis".StatusBits.HomingDone THEN
       #home_0_mode := TRUE;
       #home_3_mode := FALSE;
   END_IF;
   IF "Rotation_Axis".StatusBits.HomingDone THEN
       #home_3_mode := FALSE;
       #home_0_mode := FALSE;
   END_IF;
END_REGION

REGION Network 4: Ручная калибровка
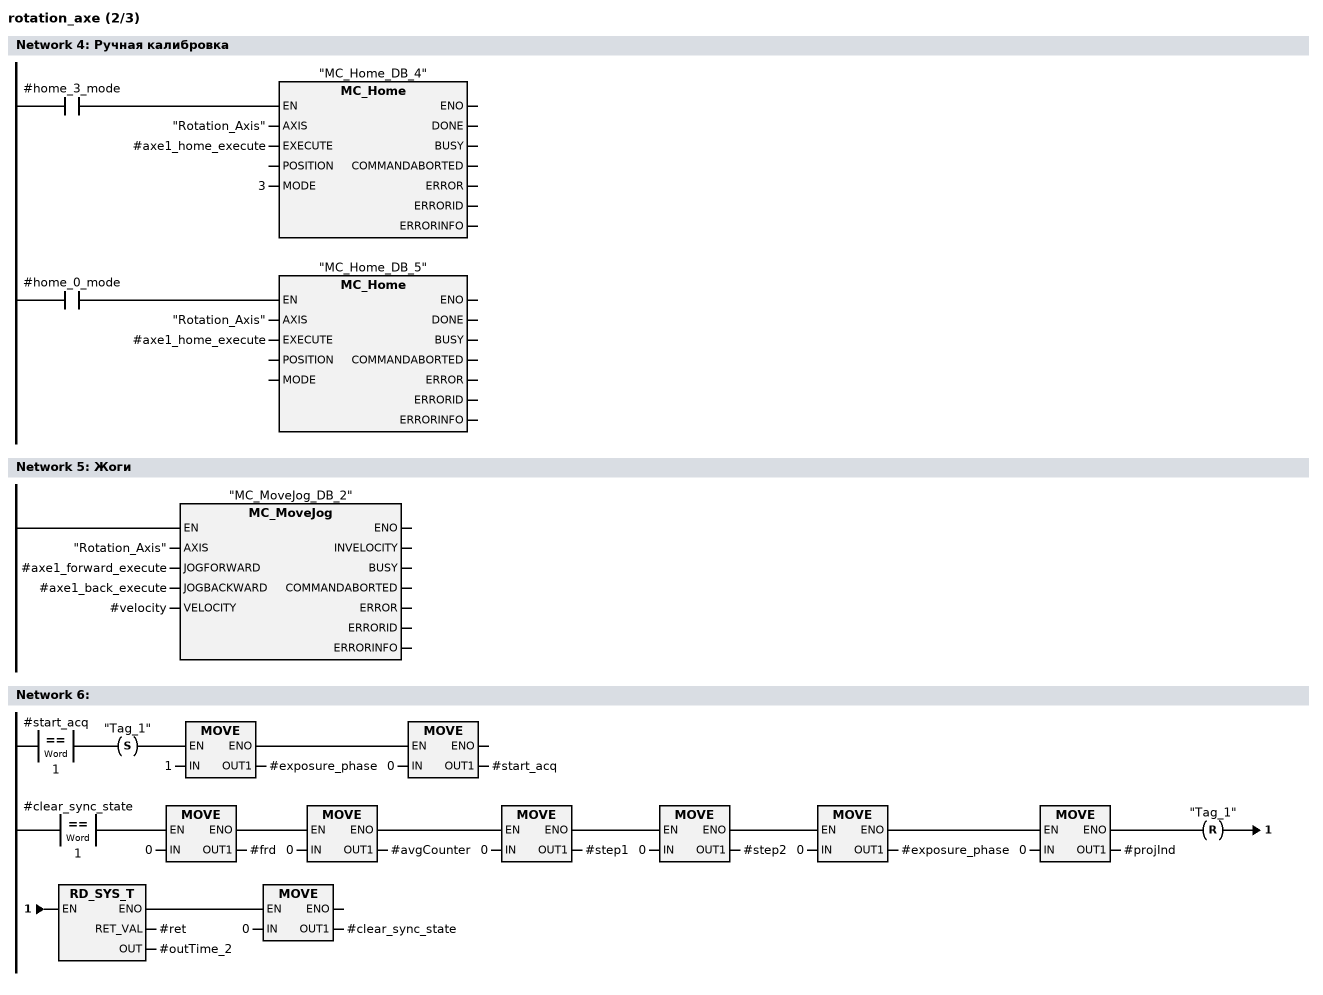
   IF #home_3_mode THEN
       "MC_Home_DB_4"(Axis := "Rotation_Axis", Execute := #axe1_home_execute, Mode := 3);   // MC_Home
   END_IF;
   IF #home_0_mode THEN
       "MC_Home_DB_5"(Axis := "Rotation_Axis", Execute := #axe1_home_execute);   // MC_Home
   END_IF;
END_REGION

REGION Network 5: Жоги
   "MC_MoveJog_DB_2"(Axis := "Rotation_Axis",   // MC_MoveJog
                     JogForward := #axe1_forward_execute,
                     JogBackward := #axe1_back_execute,
                     Velocity := #velocity);
END_REGION

REGION Network 6
   // ENO of a box is taken as its EN; it also drops when the box reports an error
   IF #start_acq = 1 THEN
       "Tag_1" := TRUE;
       #exposure_phase := 1;
       #start_acq := 0;
   END_IF;
   IF #clear_sync_state = 1 THEN
       #frd := 0;
       #avgCounter := 0;
       #step1 := 0;
       #step2 := 0;
       #exposure_phase := 0;
       #projInd := 0;
       "Tag_1" := FALSE;
       #ret := RD_SYS_T(OUT => #outTime_2);
       #clear_sync_state := 0;
   END_IF;
END_REGION

REGION Network 7
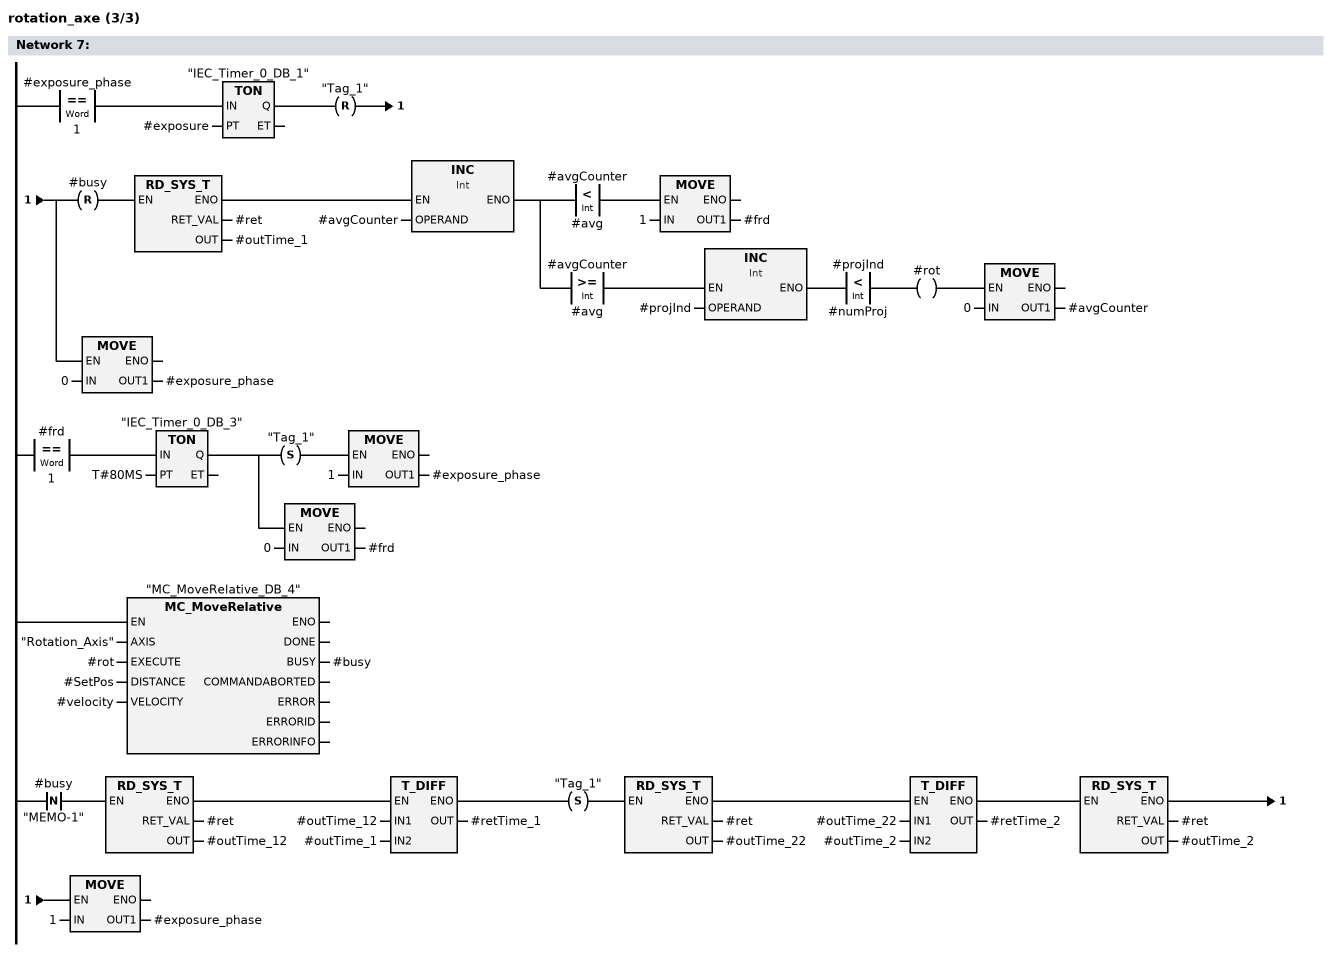
   // ENO of a box is taken as its EN; it also drops when the box reports an error
   "IEC_Timer_0_DB_1".TON(IN := #exposure_phase = 1, PT := #exposure);
   IF "IEC_Timer_0_DB_1".Q THEN
       "Tag_1" := FALSE;
       #busy := FALSE;
   END_IF;
   #_w1 := "IEC_Timer_0_DB_1".Q;
   #_w2 := "IEC_Timer_0_DB_1".Q;
   IF #_w2 THEN
       #ret := RD_SYS_T(OUT => #outTime_1);
       #avgCounter := #avgCounter + 1;
   END_IF;
   IF #_w2 AND (#avgCounter < #avg) THEN #frd := 1; END_IF;
   #_w3 := #_w2 AND (#avgCounter >= #avg);
   IF #_w3 THEN #projInd := #projInd + 1; END_IF;
   #rot := #_w3 AND (#projInd < #numProj);
   IF #rot THEN #avgCounter := 0; END_IF;
   IF #_w1 THEN #exposure_phase := 0; END_IF;
   "IEC_Timer_0_DB_3".TON(IN := #frd = 1, PT := T#80MS);
   IF "IEC_Timer_0_DB_3".Q THEN
       "Tag_1" := TRUE;
       #exposure_phase := 1;
       #frd := 0;
   END_IF;
   "MC_MoveRelative_DB_4"(Axis := "Rotation_Axis",   // MC_MoveRelative
                          Execute := #rot,
                          Distance := #SetPos,
                          Velocity := #velocity,
                          Busy => #busy);
   #_w4 := NOT #busy AND "MEMO-1";   // falling edge of #busy
   "MEMO-1" := #busy;
   IF #_w4 THEN
       #ret := RD_SYS_T(OUT => #outTime_12);
       #retTime_1 := T_DIFF(IN1 := #outTime_12, IN2 := #outTime_1);
       "Tag_1" := TRUE;
       #ret := RD_SYS_T(OUT => #outTime_22);
       #retTime_2 := T_DIFF(IN1 := #outTime_22, IN2 := #outTime_2);
       #ret := RD_SYS_T(OUT => #outTime_2);
       #exposure_phase := 1;
   END_IF;
END_REGION
END_FUNCTION_BLOCK

FUNCTION_BLOCK "detector_axe"   // FB4, LAD
{ S7_Optimized_Access := 'TRUE' }
VERSION : 0.1
   VAR
      SetPos : Real;
      velocity : Real;
      axe1_motion_enable : Bool;
      axe1_reset : Bool;
      axe1_halt : Bool;
      axe1_forward_execute : Bool;
      axe1_back_execute : Bool;
      axe1_home_execute : Bool;
      axe1_move_to_pos_execute : Bool;
      axe1_move_relative_execute : Bool;
      home_3_busy : Bool;
      home_0_busy : Bool;
      home_3_mode : Bool;
      home_0_mode : Bool;
      axe1_move_done : Bool;
      status : Bool;
      moveCounter : Word;
      moveFrame : Word;
      moveCounter2 : Int;
      delayedEx : Bool;
      first : Bool;
   END_VAR
   VAR CONSTANT
      vel_const : Real := 2.5;
   END_VAR
   VAR_TEMP   // added for the SCL form of the ladder/FBD networks
      _w1 : Bool;
      _w2 : Bool;
   END_VAR
BEGIN

REGION Network 1
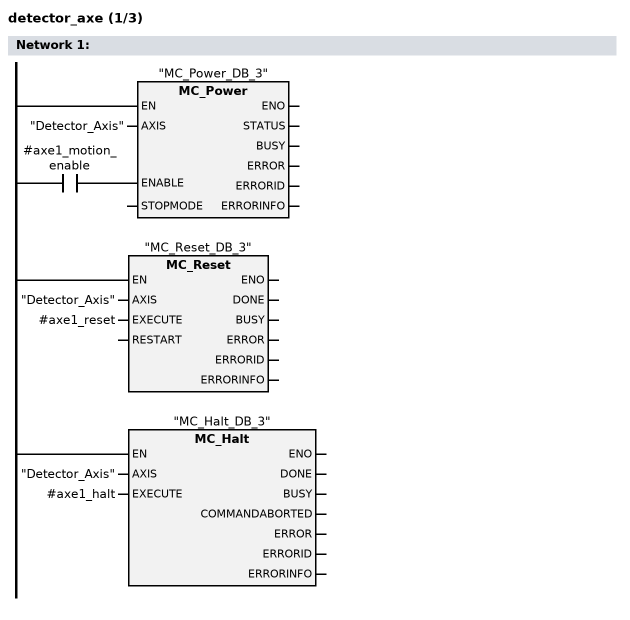
   "MC_Power_DB_3"(Axis := "Detector_Axis", Enable := #axe1_motion_enable);   // MC_Power
   "MC_Reset_DB_3"(Axis := "Detector_Axis", Execute := #axe1_reset);   // MC_Reset
   "MC_Halt_DB_3"(Axis := "Detector_Axis", Execute := #axe1_halt);   // MC_Halt
END_REGION

REGION Network 2
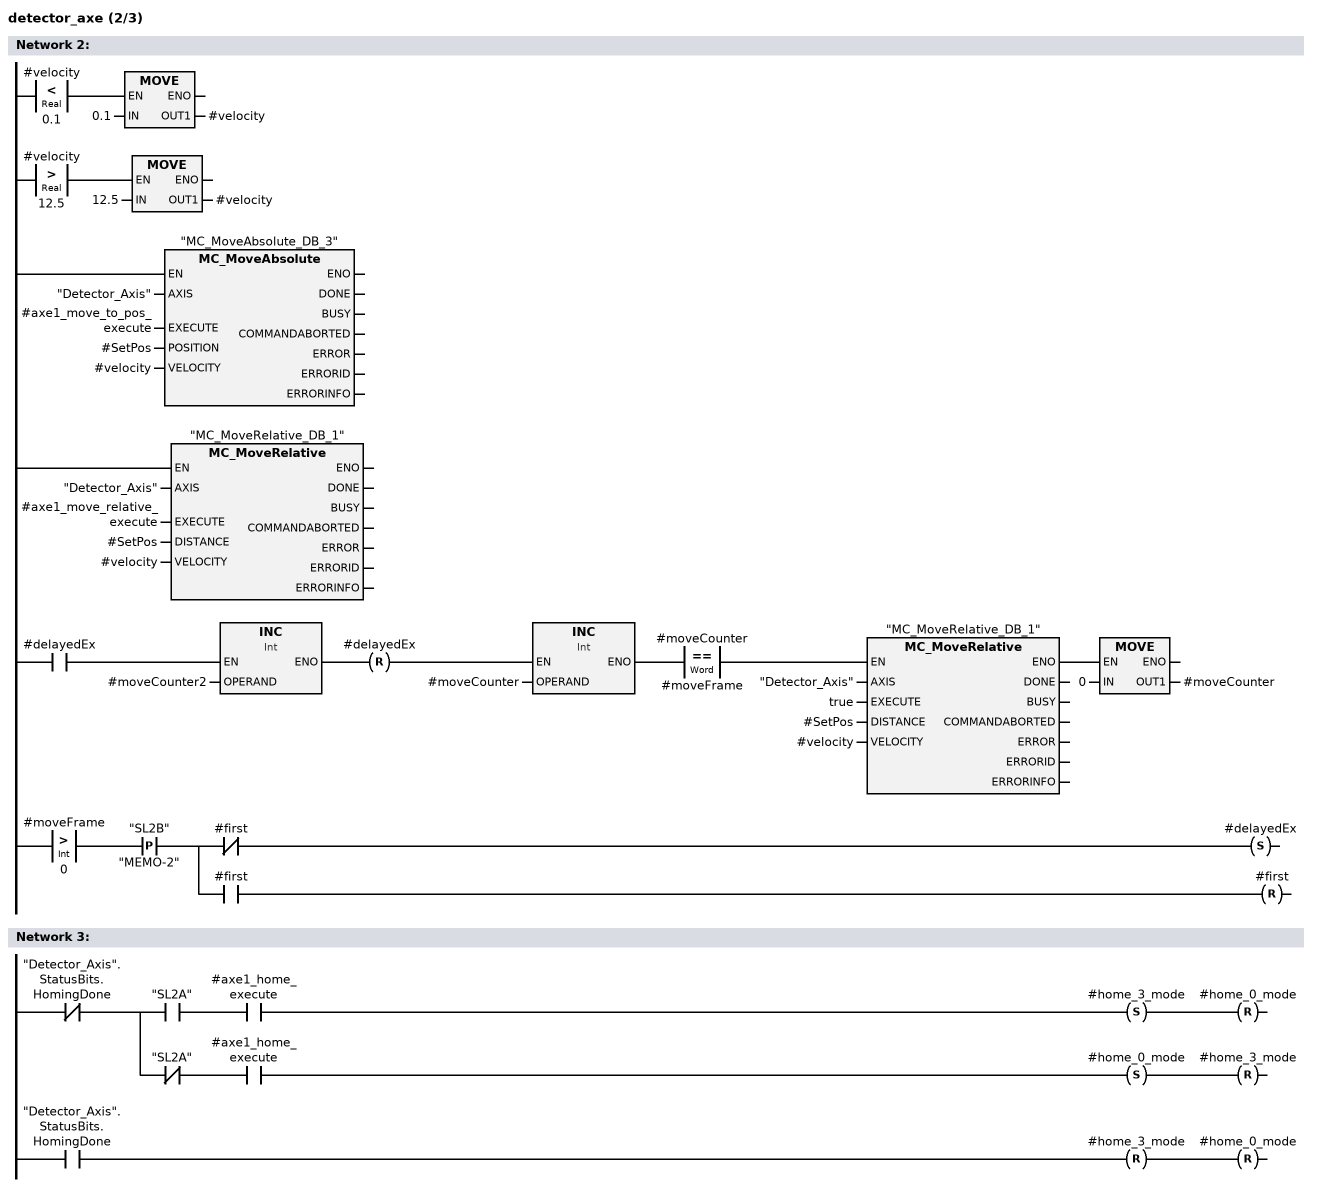
   // ENO of a box is taken as its EN; it also drops when the box reports an error
   IF #velocity < 0.1 THEN #velocity := 0.1; END_IF;
   IF #velocity > 12.5 THEN #velocity := 12.5; END_IF;
   "MC_MoveAbsolute_DB_3"(Axis := "Detector_Axis",   // MC_MoveAbsolute
                          Execute := #axe1_move_to_pos_execute,
                          Position := #SetPos,
                          Velocity := #velocity);
   "MC_MoveRelative_DB_1"(Axis := "Detector_Axis",   // MC_MoveRelative
                          Execute := #axe1_move_relative_execute,
                          Distance := #SetPos,
                          Velocity := #velocity);
   IF #delayedEx THEN #moveCounter2 := #moveCounter2 + 1; END_IF;
   #_w1 := #delayedEx;
   IF #_w1 THEN
       #delayedEx := FALSE;
       #moveCounter := #moveCounter + 1;
   END_IF;
   IF #_w1 AND (#moveCounter = #moveFrame) THEN
       "MC_MoveRelative_DB_1"(Axis := "Detector_Axis", Execute := true, Distance := #SetPos, Velocity := #velocity);   // MC_MoveRelative
       #moveCounter := 0;
   END_IF;
   #_w2 := (#moveFrame > 0) AND "SL2B" AND NOT "MEMO-2";   // rising edge of "SL2B"
   "MEMO-2" := "SL2B";
   IF #_w2 AND NOT #first THEN #delayedEx := TRUE; END_IF;
   IF #_w2 AND #first THEN #first := FALSE; END_IF;
END_REGION

REGION Network 3
   RUNG wire#powerrail
      I_Contact( "Detector_Axis".StatusBits.HomingDone )
      wire#w1
      Contact( "SL2A" )
      Contact( #axe1_home_execute )
      S_Coil( #home_3_mode )
      R_Coil( #home_0_mode )
   END_RUNG
   RUNG wire#w1
      I_Contact( "SL2A" )
      Contact( #axe1_home_execute )
      S_Coil( #home_0_mode )
      R_Coil( #home_3_mode )
   END_RUNG
   RUNG wire#powerrail
      Contact( "Detector_Axis".StatusBits.HomingDone )
      R_Coil( #home_3_mode )
      R_Coil( #home_0_mode )
   END_RUNG
   // the same network as SCL:
   #_w1 := NOT "Detector_Axis".StatusBits.HomingDone;
   IF #_w1 AND "SL2A" AND #axe1_home_execute THEN
       #home_3_mode := TRUE;
       #home_0_mode := FALSE;
   END_IF;
   IF #_w1 AND NOT "SL2A" AND #axe1_home_execute THEN
       #home_0_mode := TRUE;
       #home_3_mode := FALSE;
   END_IF;
   IF "Detector_Axis".StatusBits.HomingDone THEN
       #home_3_mode := FALSE;
       #home_0_mode := FALSE;
   END_IF;
END_REGION

REGION Network 4: Ручная калибровка
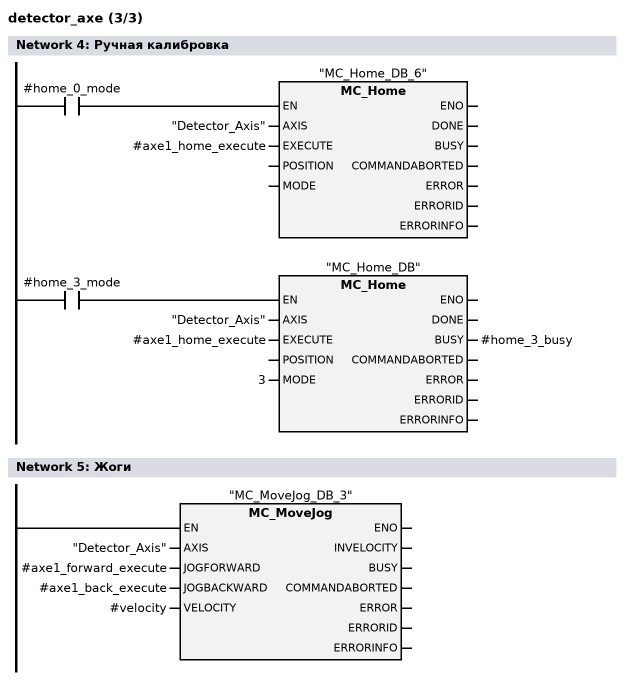
   IF #home_0_mode THEN
       "MC_Home_DB_6"(Axis := "Detector_Axis", Execute := #axe1_home_execute);   // MC_Home
   END_IF;
   IF #home_3_mode THEN
       "MC_Home_DB"(Axis := "Detector_Axis", Execute := #axe1_home_execute, Mode := 3, Busy => #home_3_busy);   // MC_Home
   END_IF;
END_REGION

REGION Network 5: Жоги
   "MC_MoveJog_DB_3"(Axis := "Detector_Axis",   // MC_MoveJog
                     JogForward := #axe1_forward_execute,
                     JogBackward := #axe1_back_execute,
                     Velocity := #velocity);
END_REGION
END_FUNCTION_BLOCK

FUNCTION_BLOCK "safety"   // FB5, LAD
{ S7_Optimized_Access := 'TRUE' }
VERSION : 0.1
BEGIN

REGION Network 1: блокировка излучекеия при открытом периметри
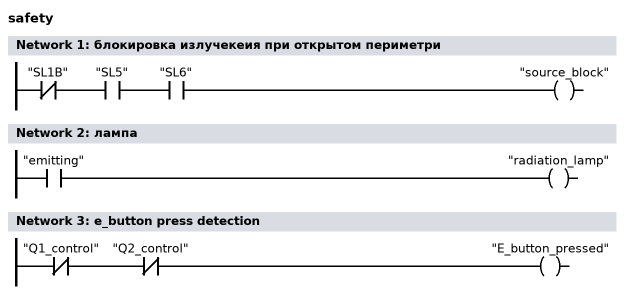
   RUNG wire#powerrail
      I_Contact( "SL1B" )
      Contact( "SL5" )
      Contact( "SL6" )
      Coil( "source_block" )
   END_RUNG
   // the same network as SCL:
   "source_block" := NOT "SL1B" AND "SL5" AND "SL6";
END_REGION

REGION Network 2: лампа
   RUNG wire#powerrail
      Contact( "emitting" )
      Coil( "radiation_lamp" )
   END_RUNG
   // the same network as SCL:
   "radiation_lamp" := "emitting";
END_REGION

REGION Network 3: e_button press detection
   RUNG wire#powerrail
      I_Contact( "Q1_control" )
      I_Contact( "Q2_control" )
      Coil( "E_button_pressed" )
   END_RUNG
   // the same network as SCL:
   "E_button_pressed" := NOT "Q1_control" AND NOT "Q2_control";
END_REGION
END_FUNCTION_BLOCK

FUNCTION_BLOCK "iso_axe"   // FB12, LAD
{ S7_Optimized_Access := 'TRUE' }
VERSION : 0.1
   VAR
      SetPos : Real;
      velocity : Real;
      axe1_motion_enable : Bool;
      axe1_reset : Bool;
      axe1_halt : Bool;
      axe1_forward_execute : Bool;
      axe1_back_execute : Bool;
      axe1_home_execute : Bool;
      axe1_move_to_pos_execute : Bool;
      axe1_move_relative_execute : Bool;
      home_3_busy : Bool;
      home_0_busy : Bool;
      home_3_mode : Bool;
      home_0_mode : Bool;
      axe1_move_done : Bool;
      status : Bool;
   END_VAR
   VAR CONSTANT
      vel_const : Real := 2.5;
   END_VAR
   VAR_TEMP   // added for the SCL form of the ladder/FBD networks
      _w1 : Bool;
   END_VAR
BEGIN

REGION Network 1
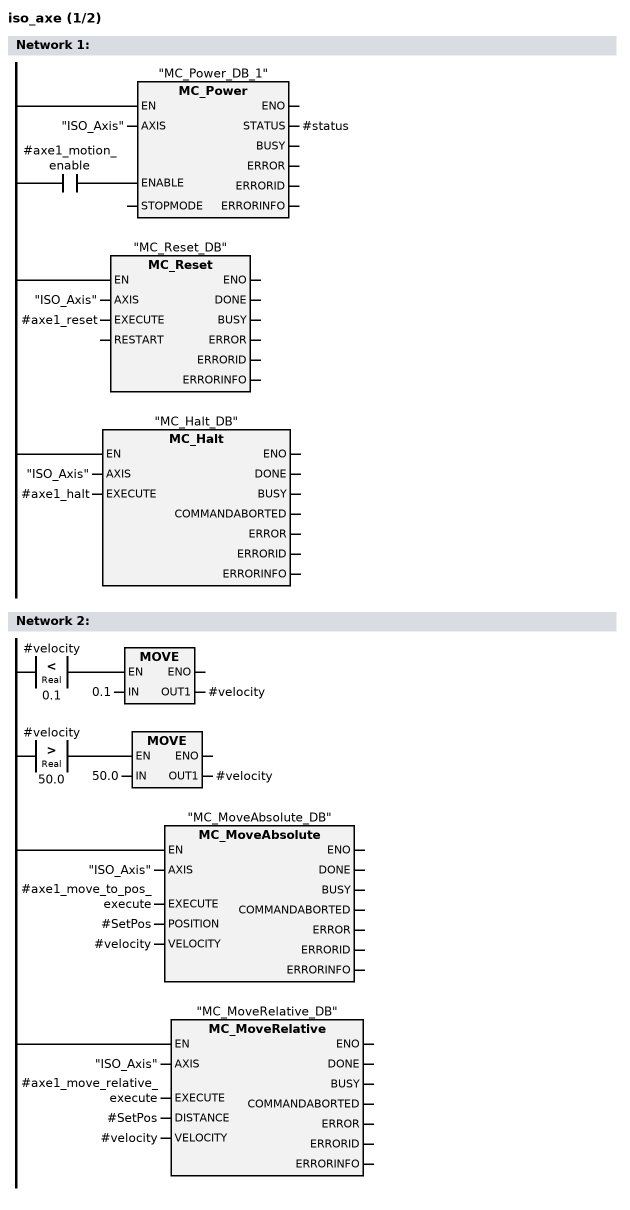
   "MC_Power_DB_1"(Axis := "ISO_Axis", Enable := #axe1_motion_enable, Status => #status);   // MC_Power
   "MC_Reset_DB"(Axis := "ISO_Axis", Execute := #axe1_reset);   // MC_Reset
   "MC_Halt_DB"(Axis := "ISO_Axis", Execute := #axe1_halt);   // MC_Halt
END_REGION

REGION Network 2
   IF #velocity < 0.1 THEN #velocity := 0.1; END_IF;
   IF #velocity > 50.0 THEN #velocity := 50.0; END_IF;
   "MC_MoveAbsolute_DB"(Axis := "ISO_Axis",   // MC_MoveAbsolute
                        Execute := #axe1_move_to_pos_execute,
                        Position := #SetPos,
                        Velocity := #velocity);
   "MC_MoveRelative_DB"(Axis := "ISO_Axis",   // MC_MoveRelative
                        Execute := #axe1_move_relative_execute,
                        Distance := #SetPos,
                        Velocity := #velocity);
END_REGION

REGION Network 3
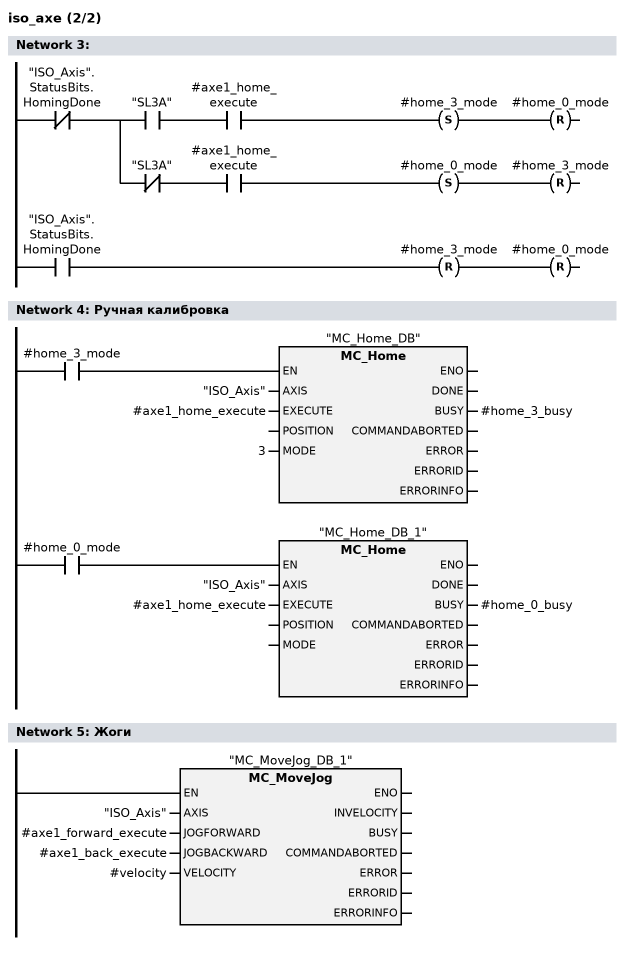
   RUNG wire#powerrail
      I_Contact( "ISO_Axis".StatusBits.HomingDone )
      wire#w1
      Contact( "SL3A" )
      Contact( #axe1_home_execute )
      S_Coil( #home_3_mode )
      R_Coil( #home_0_mode )
   END_RUNG
   RUNG wire#w1
      I_Contact( "SL3A" )
      Contact( #axe1_home_execute )
      S_Coil( #home_0_mode )
      R_Coil( #home_3_mode )
   END_RUNG
   RUNG wire#powerrail
      Contact( "ISO_Axis".StatusBits.HomingDone )
      R_Coil( #home_3_mode )
      R_Coil( #home_0_mode )
   END_RUNG
   // the same network as SCL:
   #_w1 := NOT "ISO_Axis".StatusBits.HomingDone;
   IF #_w1 AND "SL3A" AND #axe1_home_execute THEN
       #home_3_mode := TRUE;
       #home_0_mode := FALSE;
   END_IF;
   IF #_w1 AND NOT "SL3A" AND #axe1_home_execute THEN
       #home_0_mode := TRUE;
       #home_3_mode := FALSE;
   END_IF;
   IF "ISO_Axis".StatusBits.HomingDone THEN
       #home_3_mode := FALSE;
       #home_0_mode := FALSE;
   END_IF;
END_REGION

REGION Network 4: Ручная калибровка
   IF #home_3_mode THEN
       "MC_Home_DB"(Axis := "ISO_Axis", Execute := #axe1_home_execute, Mode := 3, Busy => #home_3_busy);   // MC_Home
   END_IF;
   IF #home_0_mode THEN
       "MC_Home_DB_1"(Axis := "ISO_Axis", Execute := #axe1_home_execute, Busy => #home_0_busy);   // MC_Home
   END_IF;
END_REGION

REGION Network 5: Жоги
   "MC_MoveJog_DB_1"(Axis := "ISO_Axis",   // MC_MoveJog
                     JogForward := #axe1_forward_execute,
                     JogBackward := #axe1_back_execute,
                     Velocity := #velocity);
END_REGION
END_FUNCTION_BLOCK

FUNCTION "ProcessCalibrationStatus" : Void   // FC1, LAD
{ S7_Optimized_Access := 'TRUE' }
VERSION : 0.1
BEGIN

REGION Network 1
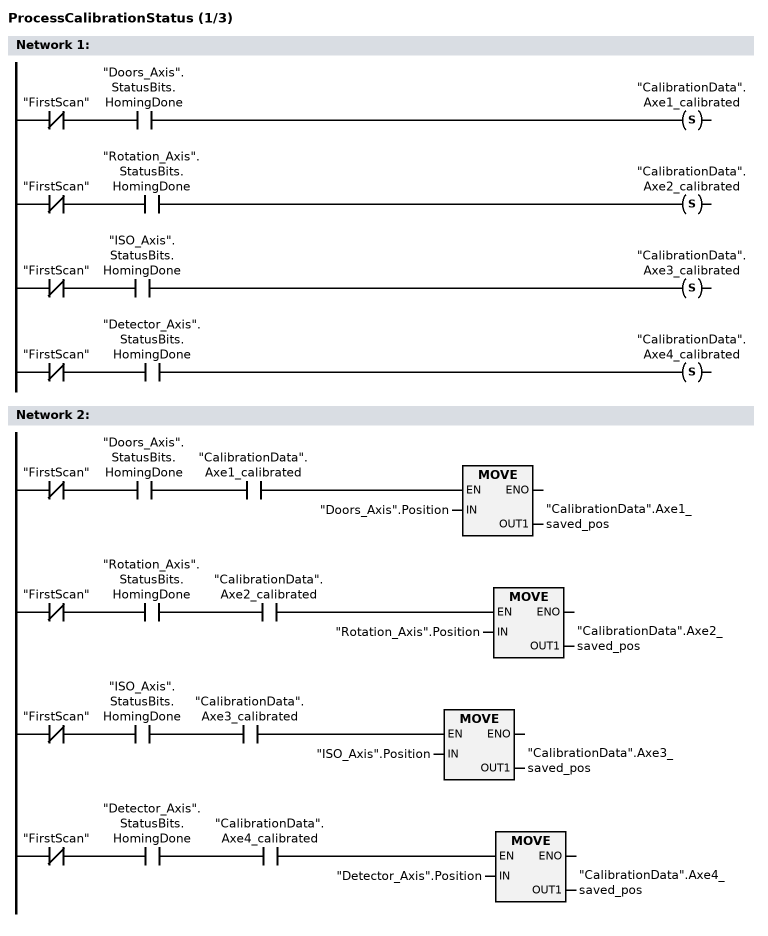
   RUNG wire#powerrail
      I_Contact( "FirstScan" )
      Contact( "Doors_Axis".StatusBits.HomingDone )
      S_Coil( "CalibrationData".Axe1_calibrated )
   END_RUNG
   RUNG wire#powerrail
      I_Contact( "FirstScan" )
      Contact( "Rotation_Axis".StatusBits.HomingDone )
      S_Coil( "CalibrationData".Axe2_calibrated )
   END_RUNG
   RUNG wire#powerrail
      I_Contact( "FirstScan" )
      Contact( "ISO_Axis".StatusBits.HomingDone )
      S_Coil( "CalibrationData".Axe3_calibrated )
   END_RUNG
   RUNG wire#powerrail
      I_Contact( "FirstScan" )
      Contact( "Detector_Axis".StatusBits.HomingDone )
      S_Coil( "CalibrationData".Axe4_calibrated )
   END_RUNG
   // the same network as SCL:
   IF NOT "FirstScan" AND "Doors_Axis".StatusBits.HomingDone THEN
       "CalibrationData".Axe1_calibrated := TRUE;
   END_IF;
   IF NOT "FirstScan" AND "Rotation_Axis".StatusBits.HomingDone THEN
       "CalibrationData".Axe2_calibrated := TRUE;
   END_IF;
   IF NOT "FirstScan" AND "ISO_Axis".StatusBits.HomingDone THEN
       "CalibrationData".Axe3_calibrated := TRUE;
   END_IF;
   IF NOT "FirstScan" AND "Detector_Axis".StatusBits.HomingDone THEN
       "CalibrationData".Axe4_calibrated := TRUE;
   END_IF;
END_REGION

REGION Network 2
   RUNG wire#powerrail
      I_Contact( "FirstScan" )
      Contact( "Doors_Axis".StatusBits.HomingDone )
      Contact( "CalibrationData".Axe1_calibrated )
      Move(in := "Doors_Axis".Position, out1 => "CalibrationData".Axe1_saved_pos)
   END_RUNG
   RUNG wire#powerrail
      I_Contact( "FirstScan" )
      Contact( "Rotation_Axis".StatusBits.HomingDone )
      Contact( "CalibrationData".Axe2_calibrated )
      Move(in := "Rotation_Axis".Position, out1 => "CalibrationData".Axe2_saved_pos)
   END_RUNG
   RUNG wire#powerrail
      I_Contact( "FirstScan" )
      Contact( "ISO_Axis".StatusBits.HomingDone )
      Contact( "CalibrationData".Axe3_calibrated )
      Move(in := "ISO_Axis".Position, out1 => "CalibrationData".Axe3_saved_pos)
   END_RUNG
   RUNG wire#powerrail
      I_Contact( "FirstScan" )
      Contact( "Detector_Axis".StatusBits.HomingDone )
      Contact( "CalibrationData".Axe4_calibrated )
      Move(in := "Detector_Axis".Position, out1 => "CalibrationData".Axe4_saved_pos)
   END_RUNG
   // the same network as SCL:
   IF NOT "FirstScan" AND "Doors_Axis".StatusBits.HomingDone AND "CalibrationData".Axe1_calibrated THEN
       "CalibrationData".Axe1_saved_pos := "Doors_Axis".Position;
   END_IF;
   IF NOT "FirstScan" AND "Rotation_Axis".StatusBits.HomingDone AND "CalibrationData".Axe2_calibrated THEN
       "CalibrationData".Axe2_saved_pos := "Rotation_Axis".Position;
   END_IF;
   IF NOT "FirstScan" AND "ISO_Axis".StatusBits.HomingDone AND "CalibrationData".Axe3_calibrated THEN
       "CalibrationData".Axe3_saved_pos := "ISO_Axis".Position;
   END_IF;
   IF NOT "FirstScan" AND "Detector_Axis".StatusBits.HomingDone AND "CalibrationData".Axe4_calibrated THEN
       "CalibrationData".Axe4_saved_pos := "Detector_Axis".Position;
   END_IF;
END_REGION

REGION Network 3
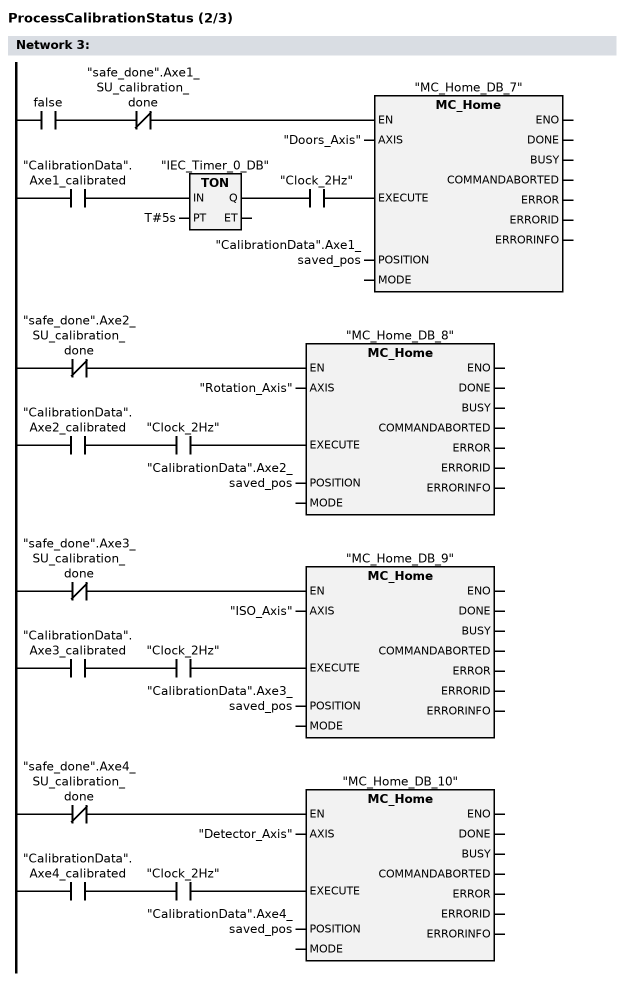
   "IEC_Timer_0_DB".TON(IN := "CalibrationData".Axe1_calibrated, PT := T#5s);
   IF false AND NOT "safe_done".Axe1_SU_calibration_done THEN
       "MC_Home_DB_7"(Axis := "Doors_Axis",   // MC_Home
                      Execute := "IEC_Timer_0_DB".Q AND "Clock_2Hz",
                      Position := "CalibrationData".Axe1_saved_pos);
   END_IF;
   IF NOT "safe_done".Axe2_SU_calibration_done THEN
       "MC_Home_DB_8"(Axis := "Rotation_Axis",   // MC_Home
                      Execute := "CalibrationData".Axe2_calibrated AND "Clock_2Hz",
                      Position := "CalibrationData".Axe2_saved_pos);
   END_IF;
   IF NOT "safe_done".Axe3_SU_calibration_done THEN
       "MC_Home_DB_9"(Axis := "ISO_Axis",   // MC_Home
                      Execute := "CalibrationData".Axe3_calibrated AND "Clock_2Hz",
                      Position := "CalibrationData".Axe3_saved_pos);
   END_IF;
   IF NOT "safe_done".Axe4_SU_calibration_done THEN
       "MC_Home_DB_10"(Axis := "Detector_Axis",   // MC_Home
                       Execute := "CalibrationData".Axe4_calibrated AND "Clock_2Hz",
                       Position := "CalibrationData".Axe4_saved_pos);
   END_IF;
END_REGION

REGION Network 4
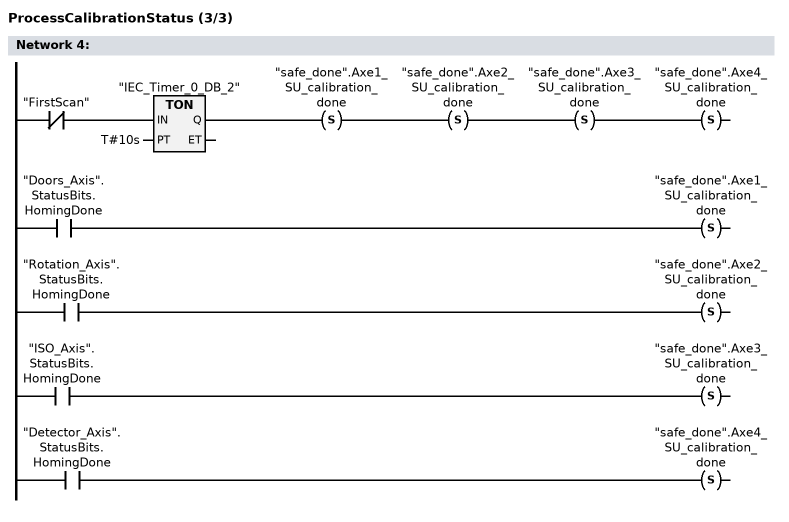
   "IEC_Timer_0_DB_2".TON(IN := NOT "FirstScan", PT := T#10s);
   IF "IEC_Timer_0_DB_2".Q THEN
       "safe_done".Axe1_SU_calibration_done := TRUE;
       "safe_done".Axe2_SU_calibration_done := TRUE;
       "safe_done".Axe3_SU_calibration_done := TRUE;
       "safe_done".Axe4_SU_calibration_done := TRUE;
   END_IF;
   IF "Doors_Axis".StatusBits.HomingDone THEN "safe_done".Axe1_SU_calibration_done := TRUE; END_IF;
   IF "Rotation_Axis".StatusBits.HomingDone THEN "safe_done".Axe2_SU_calibration_done := TRUE; END_IF;
   IF "ISO_Axis".StatusBits.HomingDone THEN "safe_done".Axe3_SU_calibration_done := TRUE; END_IF;
   IF "Detector_Axis".StatusBits.HomingDone THEN "safe_done".Axe4_SU_calibration_done := TRUE; END_IF;
END_REGION
END_FUNCTION

ORGANIZATION_BLOCK "Main"   // OB1, LAD, ProgramCycle
TITLE = "Main Program Sweep (Cycle)"
{ S7_Optimized_Access := 'TRUE' }
VERSION : 0.1
   VAR_INPUT
      Initial_Call : Bool;   // Initial call of this OB
      Remanence : Bool;   // =True, if remanent data are available
   END_VAR
BEGIN

REGION Network 1
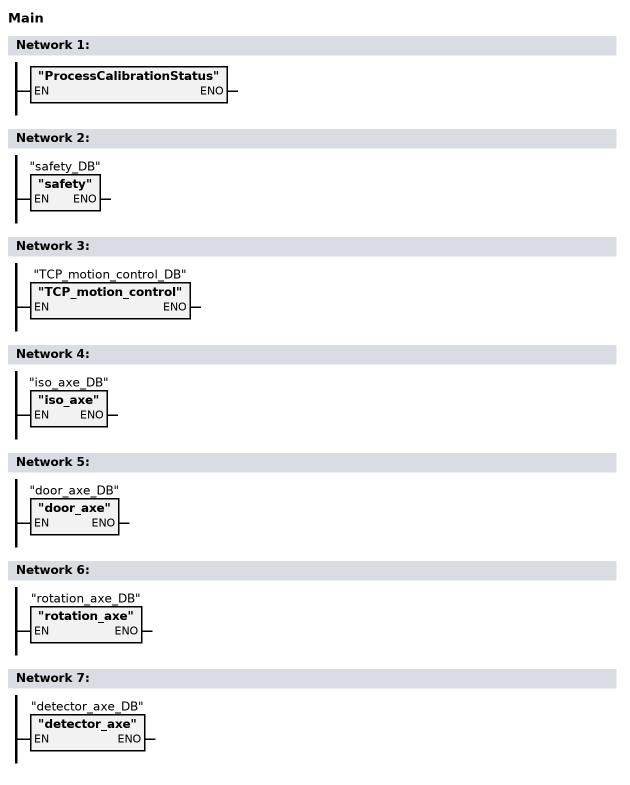
   RUNG wire#powerrail
      "ProcessCalibrationStatus"()
   END_RUNG
   // the same network as SCL:
   "ProcessCalibrationStatus"();
END_REGION

REGION Network 2
   RUNG wire#powerrail
      "safety_DB"()
   END_RUNG
   // the same network as SCL:
   "safety_DB"();   // "safety"
END_REGION

REGION Network 3
   RUNG wire#powerrail
      "TCP_motion_control_DB"()
   END_RUNG
   // the same network as SCL:
   "TCP_motion_control_DB"();   // "TCP_motion_control"
END_REGION

REGION Network 4
   RUNG wire#powerrail
      "iso_axe_DB"()
   END_RUNG
   // the same network as SCL:
   "iso_axe_DB"();   // "iso_axe"
END_REGION

REGION Network 5
   RUNG wire#powerrail
      "door_axe_DB"()
   END_RUNG
   // the same network as SCL:
   "door_axe_DB"();   // "door_axe"
END_REGION

REGION Network 6
   RUNG wire#powerrail
      "rotation_axe_DB"()
   END_RUNG
   // the same network as SCL:
   "rotation_axe_DB"();   // "rotation_axe"
END_REGION

REGION Network 7
   RUNG wire#powerrail
      "detector_axe_DB"()
   END_RUNG
   // the same network as SCL:
   "detector_axe_DB"();   // "detector_axe"
END_REGION
END_ORGANIZATION_BLOCK